LIN {X 0,Y 578.15,Z 1208.915,A -85,B 0,C 180,E1 8907.003,E2 8907.003} C_VEL
LIN {X 0,Y 578.339,Z 1209.667,A -85,B 0,C 180,E1 8911.496,E2 8911.496} C_VEL
LIN {X 0,Y 578.199,Z 1205.911,A -85,B 0,C 180,E1 8916,E2 8916} C_VEL
LIN {X 0,Y 578.472,Z 1197.323,A -85,B 0,C 180,E1 8920.535,E2 8920.535} C_VEL
LIN {X 0,Y 579.28,Z 1182.503,A -85,B 0,C 180,E1 8925.469,E2 8925.469} C_VEL
LIN {X 0,Y 580.832,Z 1163.752,A -85,B 0,C 180,E1 8929.975,E2 8929.975} C_VEL
LIN {X 0,Y 583.523,Z 1139.24,A -85,B 0,C 180,E1 8934.477,E2 8934.477} C_VEL
LIN {X 0,Y 587.576,Z 1110.062,A -85,B 0,C 180,E1 8938.727,E2 8938.727} C_VEL
LIN {X 0,Y 593,Z 1073.863,A -85,B 0,C 180,E1 8942.879,E2 8942.879} C_VEL
LIN {X 0,Y 598.958,Z 1035.476,A -85,B 0,C 180,E1 8946.381,E2 8946.381} C_VEL
LIN {X 0,Y 605.258,Z 993.744,A -85,B 0,C 180,E1 8949.361,E2 8949.361} C_VEL
LIN {X 0,Y 611.066,Z 950.98,A -85,B 0,C 180,E1 8951.738,E2 8951.738} C_VEL
LIN {X 0,Y 616.329,Z 901.945,A -85,B 0,C 180,E1 8953.734,E2 8953.734} C_VEL
LIN {X 0,Y 620.351,Z 854.304,A -85,B 0,C 180,E1 8955.052,E2 8955.052} C_VEL
LIN {X 0,Y 621.032,Z 836.384,A -85,B 0,C 180,E1 8955.439,E2 8955.439} C_VEL
LIN {X 0,Y 598.795,Z 797.154,A -85,B 0,C 180,E1 8958.388,E2 8958.388} C_VEL
LIN {X 0,Y 579.202,Z 767.417,A -85,B 0,C 180,E1 8961.172,E2 8961.172} C_VEL
LIN {X 0,Y 577.121,Z 762.06,A -85,B 0,C 180,E1 8961.632,E2 8961.632} C_VEL
LIN {X 0,Y 577.165,Z 762.06,A -85,B 0,C 180,E1 8966.908,E2 8966.908} C_VEL
LIN {X 0,Y 577.19,Z 762.06,A -85,B 0,C 180,E1 8972.889,E2 8972.889} C_VEL
LIN {X 0,Y 577.361,Z 762.06,A -85,B 0,C 180,E1 8978.499,E2 8978.499} C_VEL
LIN {X 0,Y 577.553,Z 762.06,A -85,B 0,C 180,E1 8983.267,E2 8983.267} C_VEL
LIN {X 0,Y 577.681,Z 762.06,A -85,B 0,C 180,E1 8987.913,E2 8987.913} C_VEL
LIN {X 0,Y 577.909,Z 762.06,A -85,B 0,C 180,E1 8993.988,E2 8993.988} C_VEL
LIN {X 0,Y 578.159,Z 762.06,A -85,B 0,C 180,E1 8999.991,E2 8999.991} C_VEL
LIN {X 0,Y 577.988,Z 762.06,A -85,B 0,C 180,E1 9004.489,E2 9004.489} C_VEL
LIN {X 0,Y 577.816,Z 762.06,A -85,B 0,C 180,E1 9009.018,E2 9009.018} C_VEL
LIN {X 0,Y 577.434,Z 762.06,A -85,B 0,C 180,E1 9014.476,E2 9014.476} C_VEL
LIN {X 0,Y 577.29,Z 762.06,A -85,B 0,C 180,E1 9019.882,E2 9019.882} C_VEL
LIN {X 0,Y 577.282,Z 762.06,A -85,B 0,C 180,E1 9024.747,E2 9024.747} C_VEL
LIN {X 0,Y 577.169,Z 762.06,A -85,B 0,C 180,E1 9030.234,E2 9030.234} C_VEL
LIN {X 0,Y 577.087,Z 762.06,A -85,B 0,C 180,E1 9035.735,E2 9035.735} C_VEL
LIN {X 0,Y 577.062,Z 762.06,A -85,B 0,C 180,E1 9038.874,E2 9038.874} C_VEL
LIN {X 0,Y 579.277,Z 767.544,A -85,B 0,C 180,E1 9039.257,E2 9039.257} C_VEL
LIN {X 0,Y 602.052,Z 802.935,A -85,B 0,C 180,E1 9042.524,E2 9042.524} C_VEL
LIN {X 0,Y 619.608,Z 836.668,A -85,B 0,C 180,E1 9045.179,E2 9045.179} C_VEL
LIN {X 0,Y 615.139,Z 886.033,A -85,B 0,C 180,E1 9046.707,E2 9046.707} C_VEL
LIN {X 0,Y 609.48,Z 932.606,A -85,B 0,C 180,E1 9048.803,E2 9048.803} C_VEL
LIN {X 0,Y 603.473,Z 975.898,A -85,B 0,C 180,E1 9051.376,E2 9051.376} C_VEL
LIN {X 0,Y 597.201,Z 1016.98,A -85,B 0,C 180,E1 9054.547,E2 9054.547} C_VEL
LIN {X 0,Y 591.368,Z 1054.56,A -85,B 0,C 180,E1 9058.196,E2 9058.196} C_VEL
LIN {X 0,Y 586.176,Z 1089.448,A -85,B 0,C 180,E1 9062.497,E2 9062.497} C_VEL
LIN {X 0,Y 582.691,Z 1117.096,A -85,B 0,C 180,E1 9066.804,E2 9066.804} C_VEL
LIN {X 0,Y 580.137,Z 1141.903,A -85,B 0,C 180,E1 9071.787,E2 9071.787} C_VEL
LIN {X 0,Y 578.907,Z 1159.014,A -85,B 0,C 180,E1 9076.414,E2 9076.414} C_VEL
LIN {X 0,Y 578.272,Z 1170.777,A -85,B 0,C 180,E1 9080.98,E2 9080.98} C_VEL
LIN {X 0,Y 578.016,Z 1177.724,A -85,B 0,C 180,E1 9085.502,E2 9085.502} C_VEL
LIN {X 0,Y 578.08,Z 1179.996,A -85,B 0,C 180,E1 9090.001,E2 9090.001} C_VEL
LIN {X 0,Y 578.131,Z 1177.619,A -85,B 0,C 180,E1 9094.498,E2 9094.498} C_VEL
LIN {X 0,Y 578.336,Z 1170.588,A -85,B 0,C 180,E1 9099.02,E2 9099.02} C_VEL
LIN {X 0,Y 578.842,Z 1158.74,A -85,B 0,C 180,E1 9103.59,E2 9103.59} C_VEL
LIN {X 0,Y 580.096,Z 1141.5,A -85,B 0,C 180,E1 9108.216,E2 9108.216} C_VEL
LIN {X 0,Y 582.461,Z 1118.253,A -85,B 0,C 180,E1 9112.903,E2 9112.903} C_VEL
LIN {X 0,Y 586.041,Z 1090.589,A -85,B 0,C 180,E1 9117.256,E2 9117.256} C_VEL
LIN {X 0,Y 591.234,Z 1055.571,A -85,B 0,C 180,E1 9121.599,E2 9121.599} C_VEL
LIN {X 0,Y 596.909,Z 1018.606,A -85,B 0,C 180,E1 9125.225,E2 9125.225} C_VEL
LIN {X 0,Y 603.422,Z 976.128,A -85,B 0,C 180,E1 9128.518,E2 9128.518} C_VEL
LIN {X 0,Y 609.637,Z 932.43,A -85,B 0,C 180,E1 9131.105,E2 9131.105} C_VEL
LIN {X 0,Y 614.684,Z 890.546,A -85,B 0,C 180,E1 9133.017,E2 9133.017} C_VEL
LIN {X 0,Y 619.052,Z 844.789,A -85,B 0,C 180,E1 9134.528,E2 9134.528} C_VEL
LIN {X 0,Y 619.221,Z 836.103,A -85,B 0,C 180,E1 9134.785,E2 9134.785} C_VEL
LIN {X 0,Y 600.743,Z 800.765,A -85,B 0,C 180,E1 9137.568,E2 9137.568} C_VEL
LIN {X 0,Y 579.4,Z 767.603,A -85,B 0,C 180,E1 9140.634,E2 9140.634} C_VEL
LIN {X 0,Y 577.111,Z 762.06,A -85,B 0,C 180,E1 9141.084,E2 9141.084} C_VEL
LIN {X 0,Y 577.121,Z 762.06,A -85,B 0,C 180,E1 9146.918,E2 9146.918} C_VEL
LIN {X 0,Y 577.114,Z 762.06,A -85,B 0,C 180,E1 9152.907,E2 9152.907} C_VEL
LIN {X 0,Y 577.261,Z 762.06,A -85,B 0,C 180,E1 9158.513,E2 9158.513} C_VEL
LIN {X 0,Y 577.429,Z 762.06,A -85,B 0,C 180,E1 9164.84,E2 9164.84} C_VEL
LIN {X 0,Y 577.724,Z 762.06,A -85,B 0,C 180,E1 9169.46,E2 9169.46} C_VEL
LIN {X 0,Y 577.901,Z 762.06,A -85,B 0,C 180,E1 9174.006,E2 9174.006} C_VEL
LIN {X 0,Y 578.06,Z 762.06,A -85,B 0,C 180,E1 9178.511,E2 9178.511} C_VEL
LIN {X 0,Y 577.954,Z 762.06,A -85,B 0,C 180,E1 9183.006,E2 9183.006} C_VEL
LIN {X 0,Y 577.846,Z 762.06,A -85,B 0,C 180,E1 9187.521,E2 9187.521} C_VEL
LIN {X 0,Y 577.677,Z 762.06,A -85,B 0,C 180,E1 9192.087,E2 9192.087} C_VEL
LIN {X 0,Y 577.633,Z 762.06,A -85,B 0,C 180,E1 9196.731,E2 9196.731} C_VEL
LIN {X 0,Y 577.501,Z 762.06,A -85,B 0,C 180,E1 9201.496,E2 9201.496} C_VEL
LIN {X 0,Y 577.334,Z 762.06,A -85,B 0,C 180,E1 9207.136,E2 9207.136} C_VEL
LIN {X 0,Y 577.241,Z 762.06,A -85,B 0,C 180,E1 9213.1,E2 9213.1} C_VEL
LIN {X 0,Y 577.123,Z 762.06,A -85,B 0,C 180,E1 9218.461,E2 9218.461} C_VEL
LIN {X 0,Y 579.443,Z 767.642,A -85,B 0,C 180,E1 9218.865,E2 9218.865} C_VEL
LIN {X 0,Y 602.931,Z 803.858,A -85,B 0,C 180,E1 9222.165,E2 9222.165} C_VEL
LIN {X 0,Y 621.477,Z 837.132,A -85,B 0,C 180,E1 9224.621,E2 9224.621} C_VEL
LIN {X 0,Y 617.556,Z 889.111,A -85,B 0,C 180,E1 9225.855,E2 9225.855} C_VEL
LIN {X 0,Y 613.175,Z 933.192,A -85,B 0,C 180,E1 9227.456,E2 9227.456} C_VEL
LIN {X 0,Y 611.803,Z 944.782,A -85,B 0,C 180,E1 9227.982,E2 9227.982} C_VEL
LIN {X 0,Y 607.308,Z 955.564,A -85,B 0,C 180,E1 9228.234,E2 9228.234} C_VEL
LIN {X 0,Y 602.903,Z 965.984,A -85,B 0,C 180,E1 9228.523,E2 9228.523} C_VEL
LIN {X 0,Y 596.636,Z 1008.633,A -85,B 0,C 180,E1 9231.126,E2 9231.126} C_VEL
LIN {X 0,Y 589.947,Z 1050.374,A -85,B 0,C 180,E1 9234.424,E2 9234.424} C_VEL
LIN {X 0,Y 584.112,Z 1085.938,A -85,B 0,C 180,E1 9237.971,E2 9237.971} C_VEL
LIN {X 0,Y 578.634,Z 1121.078,A -85,B 0,C 180,E1 9242.391,E2 9242.391} C_VEL
LIN {X 0,Y 574.815,Z 1149.399,A -85,B 0,C 180,E1 9246.946,E2 9246.946} C_VEL
LIN {X 0,Y 572.456,Z 1171.697,A -85,B 0,C 180,E1 9251.532,E2 9251.532} C_VEL
LIN {X 0,Y 571.07,Z 1188.871,A -85,B 0,C 180,E1 9256.222,E2 9256.222} C_VEL
LIN {X 0,Y 570.409,Z 1200.678,A -85,B 0,C 180,E1 9260.853,E2 9260.853} C_VEL
LIN {X 0,Y 570.191,Z 1207.667,A -85,B 0,C 180,E1 9265.439,E2 9265.439} C_VEL
LIN {X 0,Y 570.292,Z 1210,A -85,B 0,C 180,E1 9269.999,E2 9269.999} C_VEL
LIN {X 0,Y 570.191,Z 1207.67,A -85,B 0,C 180,E1 9274.559,E2 9274.559} C_VEL
LIN {X 0,Y 570.399,Z 1200.681,A -85,B 0,C 180,E1 9279.145,E2 9279.145} C_VEL
LIN {X 0,Y 571.01,Z 1188.877,A -85,B 0,C 180,E1 9283.778,E2 9283.778} C_VEL
LIN {X 0,Y 572.488,Z 1171.703,A -85,B 0,C 180,E1 9288.465,E2 9288.465} C_VEL
LIN {X 0,Y 575.129,Z 1147.41,A -85,B 0,C 180,E1 9293.415,E2 9293.415} C_VEL
LIN {X 0,Y 578.901,Z 1119.586,A -85,B 0,C 180,E1 9297.812,E2 9297.812} C_VEL
LIN {X 0,Y 584.473,Z 1084.193,A -85,B 0,C 180,E1 9302.224,E2 9302.224} C_VEL
LIN {X 0,Y 590.602,Z 1046.177,A -85,B 0,C 180,E1 9305.943,E2 9305.943} C_VEL
LIN {X 0,Y 597.246,Z 1004.955,A -85,B 0,C 180,E1 9309.134,E2 9309.134} C_VEL
LIN {X 0,Y 603.585,Z 960.631,A -85,B 0,C 180,E1 9311.754,E2 9311.754} C_VEL
LIN {X 0,Y 609.331,Z 913.705,A -85,B 0,C 180,E1 9313.837,E2 9313.837} C_VEL
LIN {X 0,Y 613.929,Z 864.169,A -85,B 0,C 180,E1 9315.339,E2 9315.339} C_VEL
LIN {X 0,Y 615.156,Z 839.358,A -85,B 0,C 180,E1 9315.914,E2 9315.914} C_VEL
LIN {X 0,Y 593.425,Z 801.025,A -85,B 0,C 180,E1 9318.901,E2 9318.901} C_VEL
LIN {X 0,Y 571.54,Z 767.635,A -85,B 0,C 180,E1 9322.125,E2 9322.125} C_VEL
LIN {X 0,Y 569.331,Z 763.533,A -85,B 0,C 180,E1 9322.492,E2 9322.492} C_VEL
LIN {X 0,Y 569.194,Z 762.06,A -85,B 0,C 180,E1 9322.602,E2 9322.602} C_VEL
LIN {X 0,Y 569.21,Z 762.06,A -85,B 0,C 180,E1 9328.158,E2 9328.158} C_VEL
LIN {X 0,Y 569.312,Z 762.06,A -85,B 0,C 180,E1 9333.171,E2 9333.171} C_VEL
LIN {X 0,Y 569.438,Z 762.06,A -85,B 0,C 180,E1 9338.245,E2 9338.245} C_VEL
LIN {X 0,Y 569.61,Z 762.06,A -85,B 0,C 180,E1 9343.026,E2 9343.026} C_VEL
LIN {X 0,Y 569.8,Z 762.06,A -85,B 0,C 180,E1 9348.881,E2 9348.881} C_VEL
LIN {X 0,Y 570.008,Z 762.06,A -85,B 0,C 180,E1 9353.905,E2 9353.905} C_VEL
LIN {X 0,Y 570.259,Z 762.06,A -85,B 0,C 180,E1 9359.991,E2 9359.991} C_VEL
LIN {X 0,Y 570.078,Z 762.06,A -85,B 0,C 180,E1 9364.552,E2 9364.552} C_VEL
LIN {X 0,Y 569.891,Z 762.06,A -85,B 0,C 180,E1 9369.144,E2 9369.144} C_VEL
LIN {X 0,Y 569.572,Z 762.06,A -85,B 0,C 180,E1 9373.803,E2 9373.803} C_VEL
LIN {X 0,Y 569.365,Z 762.06,A -85,B 0,C 180,E1 9380.171,E2 9380.171} C_VEL
LIN {X 0,Y 569.319,Z 762.06,A -85,B 0,C 180,E1 9385.521,E2 9385.521} C_VEL
LIN {X 0,Y 569.271,Z 762.06,A -85,B 0,C 180,E1 9390.274,E2 9390.274} C_VEL
LIN {X 0,Y 569.204,Z 762.06,A -85,B 0,C 180,E1 9395.72,E2 9395.72} C_VEL
LIN {X 0,Y 569.19,Z 762.554,A -85,B 0,C 180,E1 9397.887,E2 9397.887} C_VEL
LIN {X 0,Y 571.828,Z 767.957,A -85,B 0,C 180,E1 9398.335,E2 9398.335} C_VEL
LIN {X 0,Y 595.395,Z 804.724,A -85,B 0,C 180,E1 9401.853,E2 9401.853} C_VEL
LIN {X 0,Y 613.798,Z 839.794,A -85,B 0,C 180,E1 9404.73,E2 9404.73} C_VEL
LIN {X 0,Y 609.147,Z 887.831,A -85,B 0,C 180,E1 9406.252,E2 9406.252} C_VEL
LIN {X 0,Y 603.148,Z 935.142,A -85,B 0,C 180,E1 9408.424,E2 9408.424} C_VEL
LIN {X 0,Y 596.582,Z 979.085,A -85,B 0,C 180,E1 9411.114,E2 9411.114} C_VEL
LIN {X 0,Y 589.91,Z 1020.817,A -85,B 0,C 180,E1 9414.42,E2 9414.42} C_VEL
LIN {X 0,Y 584.051,Z 1056.311,A -85,B 0,C 180,E1 9417.969,E2 9417.969} C_VEL
LIN {X 0,Y 578.578,Z 1091.32,A -85,B 0,C 180,E1 9422.378,E2 9422.378} C_VEL
LIN {X 0,Y 574.813,Z 1119.4,A -85,B 0,C 180,E1 9426.902,E2 9426.902} C_VEL
LIN {X 0,Y 572.368,Z 1141.898,A -85,B 0,C 180,E1 9431.531,E2 9431.531} C_VEL
LIN {X 0,Y 571.071,Z 1159.009,A -85,B 0,C 180,E1 9436.223,E2 9436.223} C_VEL
LIN {X 0,Y 570.386,Z 1170.772,A -85,B 0,C 180,E1 9440.854,E2 9440.854} C_VEL
LIN {X 0,Y 570.117,Z 1177.721,A -85,B 0,C 180,E1 9445.44,E2 9445.44} C_VEL
LIN {X 0,Y 570.179,Z 1179.997,A -85,B 0,C 180,E1 9450.001,E2 9450.001} C_VEL
LIN {X 0,Y 570.228,Z 1177.617,A -85,B 0,C 180,E1 9454.561,E2 9454.561} C_VEL
LIN {X 0,Y 570.439,Z 1170.586,A -85,B 0,C 180,E1 9459.146,E2 9459.146} C_VEL
LIN {X 0,Y 570.998,Z 1158.739,A -85,B 0,C 180,E1 9463.78,E2 9463.78} C_VEL
LIN {X 0,Y 572.335,Z 1141.502,A -85,B 0,C 180,E1 9468.472,E2 9468.472} C_VEL
LIN {X 0,Y 574.916,Z 1118.255,A -85,B 0,C 180,E1 9473.221,E2 9473.221} C_VEL
LIN {X 0,Y 578.709,Z 1090.582,A -85,B 0,C 180,E1 9477.632,E2 9477.632} C_VEL
LIN {X 0,Y 584.177,Z 1055.584,A -85,B 0,C 180,E1 9482.024,E2 9482.024} C_VEL
LIN {X 0,Y 590.194,Z 1018.686,A -85,B 0,C 180,E1 9485.679,E2 9485.679} C_VEL
LIN {X 0,Y 597.13,Z 975.473,A -85,B 0,C 180,E1 9489.056,E2 9489.056} C_VEL
LIN {X 0,Y 604.016,Z 929.667,A -85,B 0,C 180,E1 9491.762,E2 9491.762} C_VEL
LIN {X 0,Y 609.202,Z 888.326,A -85,B 0,C 180,E1 9493.627,E2 9493.627} C_VEL
LIN {X 0,Y 613.553,Z 843.309,A -85,B 0,C 180,E1 9495.091,E2 9495.091} C_VEL
LIN {X 0,Y 612.912,Z 838.347,A -85,B 0,C 180,E1 9495.312,E2 9495.312} C_VEL
LIN {X 0,Y 594.638,Z 803.185,A -85,B 0,C 180,E1 9498.172,E2 9498.172} C_VEL
LIN {X 0,Y 571.59,Z 767.719,A -85,B 0,C 180,E1 9501.605,E2 9501.605} C_VEL
LIN {X 0,Y 569.246,Z 763.044,A -85,B 0,C 180,E1 9502.001,E2 9502.001} C_VEL
LIN {X 0,Y 569.185,Z 762.06,A -85,B 0,C 180,E1 9502.074,E2 9502.074} C_VEL
LIN {X 0,Y 569.212,Z 762.06,A -85,B 0,C 180,E1 9508.161,E2 9508.161} C_VEL
LIN {X 0,Y 569.234,Z 762.06,A -85,B 0,C 180,E1 9513.187,E2 9513.187} C_VEL
LIN {X 0,Y 569.337,Z 762.06,A -85,B 0,C 180,E1 9518.275,E2 9518.275} C_VEL
LIN {X 0,Y 569.488,Z 762.06,A -85,B 0,C 180,E1 9524.624,E2 9524.624} C_VEL
LIN {X 0,Y 569.797,Z 762.06,A -85,B 0,C 180,E1 9529.312,E2 9529.312} C_VEL
LIN {X 0,Y 570.004,Z 762.06,A -85,B 0,C 180,E1 9533.922,E2 9533.922} C_VEL
LIN {X 0,Y 570.161,Z 762.06,A -85,B 0,C 180,E1 9538.49,E2 9538.49} C_VEL
LIN {X 0,Y 570.059,Z 762.06,A -85,B 0,C 180,E1 9543.047,E2 9543.047} C_VEL
LIN {X 0,Y 569.928,Z 762.06,A -85,B 0,C 180,E1 9547.626,E2 9547.626} C_VEL
LIN {X 0,Y 569.78,Z 762.06,A -85,B 0,C 180,E1 9552.257,E2 9552.257} C_VEL
LIN {X 0,Y 569.678,Z 762.06,A -85,B 0,C 180,E1 9557.266,E2 9557.266} C_VEL
LIN {X 0,Y 569.57,Z 762.06,A -85,B 0,C 180,E1 9561.81,E2 9561.81} C_VEL
LIN {X 0,Y 569.451,Z 762.06,A -85,B 0,C 180,E1 9566.822,E2 9566.822} C_VEL
LIN {X 0,Y 569.317,Z 762.06,A -85,B 0,C 180,E1 9572.069,E2 9572.069} C_VEL
LIN {X 0,Y 569.213,Z 762.06,A -85,B 0,C 180,E1 9577.457,E2 9577.457} C_VEL
LIN {X 0,Y 571.505,Z 767.645,A -85,B 0,C 180,E1 9577.876,E2 9577.876} C_VEL
LIN {X 0,Y 593.706,Z 801.317,A -85,B 0,C 180,E1 9581.136,E2 9581.136} C_VEL
LIN {X 0,Y 615.726,Z 840.508,A -85,B 0,C 180,E1 9584.169,E2 9584.169} C_VEL
LIN {X 0,Y 611.568,Z 891.855,A -85,B 0,C 180,E1 9585.422,E2 9585.422} C_VEL
LIN {X 0,Y 606.66,Z 937.336,A -85,B 0,C 180,E1 9587.138,E2 9587.138} C_VEL
LIN {X 0,Y 602.903,Z 965.984,A -85,B 0,C 180,E1 9588.523,E2 9588.523} C_VEL
LIN {X 0,Y 597.769,Z 981.415,A -85,B 0,C 180,E1 9589.145,E2 9589.145} C_VEL
LIN {X 0,Y 592.262,Z 996.481,A -85,B 0,C 180,E1 9589.825,E2 9589.825} C_VEL
LIN {X 0,Y 585.642,Z 1036.578,A -85,B 0,C 180,E1 9592.756,E2 9592.756} C_VEL
LIN {X 0,Y 579.041,Z 1074.678,A -85,B 0,C 180,E1 9596.319,E2 9596.319} C_VEL
LIN {X 0,Y 573.096,Z 1110.074,A -85,B 0,C 180,E1 9600.478,E2 9600.478} C_VEL
LIN {X 0,Y 568.321,Z 1140.428,A -85,B 0,C 180,E1 9605.032,E2 9605.032} C_VEL
LIN {X 0,Y 565.359,Z 1164.734,A -85,B 0,C 180,E1 9609.667,E2 9609.667} C_VEL
LIN {X 0,Y 563.548,Z 1183.702,A -85,B 0,C 180,E1 9614.445,E2 9614.445} C_VEL
LIN {X 0,Y 562.737,Z 1197.314,A -85,B 0,C 180,E1 9619.165,E2 9619.165} C_VEL
LIN {X 0,Y 562.409,Z 1205.908,A -85,B 0,C 180,E1 9623.829,E2 9623.829} C_VEL
LIN {X 0,Y 562.268,Z 1209.666,A -85,B 0,C 180,E1 9628.459,E2 9628.459} C_VEL
LIN {X 0,Y 562.401,Z 1208.911,A -85,B 0,C 180,E1 9633.08,E2 9633.08} C_VEL
LIN {X 0,Y 562.433,Z 1203.551,A -85,B 0,C 180,E1 9637.72,E2 9637.72} C_VEL
LIN {X 0,Y 562.835,Z 1193.421,A -85,B 0,C 180,E1 9642.402,E2 9642.402} C_VEL
LIN {X 0,Y 564.018,Z 1178.003,A -85,B 0,C 180,E1 9647.139,E2 9647.139} C_VEL
LIN {X 0,Y 566.256,Z 1156.978,A -85,B 0,C 180,E1 9651.937,E2 9651.937} C_VEL
LIN {X 0,Y 569.716,Z 1131.625,A -85,B 0,C 180,E1 9656.402,E2 9656.402} C_VEL
LIN {X 0,Y 574.953,Z 1099.018,A -85,B 0,C 180,E1 9660.925,E2 9660.925} C_VEL
LIN {X 0,Y 580.878,Z 1063.701,A -85,B 0,C 180,E1 9664.797,E2 9664.797} C_VEL
LIN {X 0,Y 587.848,Z 1023.085,A -85,B 0,C 180,E1 9668.326,E2 9668.326} C_VEL
LIN {X 0,Y 594.574,Z 981.096,A -85,B 0,C 180,E1 9671.128,E2 9671.128} C_VEL
LIN {X 0,Y 600.97,Z 935.912,A -85,B 0,C 180,E1 9673.434,E2 9673.434} C_VEL
LIN {X 0,Y 605.868,Z 892.707,A -85,B 0,C 180,E1 9675.069,E2 9675.069} C_VEL
LIN {X 0,Y 609.423,Z 842.612,A -85,B 0,C 180,E1 9676.382,E2 9676.382} C_VEL
LIN {X 0,Y 587.325,Z 803.329,A -85,B 0,C 180,E1 9679.54,E2 9679.54} C_VEL
LIN {X 0,Y 563.946,Z 767.982,A -85,B 0,C 180,E1 9683.113,E2 9683.113} C_VEL
LIN {X 0,Y 561.288,Z 762.651,A -85,B 0,C 180,E1 9683.585,E2 9683.585} C_VEL
LIN {X 0,Y 561.297,Z 762.06,A -85,B 0,C 180,E1 9689.484,E2 9689.484} C_VEL
LIN {X 0,Y 561.426,Z 762.06,A -85,B 0,C 180,E1 9694.485,E2 9694.485} C_VEL
LIN {X 0,Y 561.574,Z 762.06,A -85,B 0,C 180,E1 9700.353,E2 9700.353} C_VEL
LIN {X 0,Y 561.786,Z 762.06,A -85,B 0,C 180,E1 9705.983,E2 9705.983} C_VEL
LIN {X 0,Y 561.943,Z 762.06,A -85,B 0,C 180,E1 9710.707,E2 9710.707} C_VEL
LIN {X 0,Y 562.162,Z 762.06,A -85,B 0,C 180,E1 9715.366,E2 9715.366} C_VEL
LIN {X 0,Y 562.358,Z 762.06,A -85,B 0,C 180,E1 9719.991,E2 9719.991} C_VEL
LIN {X 0,Y 562.167,Z 762.06,A -85,B 0,C 180,E1 9724.616,E2 9724.616} C_VEL
LIN {X 0,Y 561.976,Z 762.06,A -85,B 0,C 180,E1 9729.274,E2 9729.274} C_VEL
LIN {X 0,Y 561.615,Z 762.06,A -85,B 0,C 180,E1 9734.391,E2 9734.391} C_VEL
LIN {X 0,Y 561.457,Z 762.06,A -85,B 0,C 180,E1 9740.468,E2 9740.468} C_VEL
LIN {X 0,Y 561.437,Z 762.06,A -85,B 0,C 180,E1 9745.495,E2 9745.495} C_VEL
LIN {X 0,Y 561.345,Z 762.06,A -85,B 0,C 180,E1 9750.747,E2 9750.747} C_VEL
LIN {X 0,Y 561.271,Z 762.06,A -85,B 0,C 180,E1 9756.804,E2 9756.804} C_VEL
LIN {X 0,Y 563.465,Z 767.461,A -85,B 0,C 180,E1 9757.228,E2 9757.228} C_VEL
LIN {X 0,Y 584.428,Z 799.083,A -85,B 0,C 180,E1 9760.503,E2 9760.503} C_VEL
LIN {X 0,Y 605.427,Z 837.685,A -85,B 0,C 180,E1 9763.843,E2 9763.843} C_VEL
LIN {X 0,Y 607.975,Z 843.781,A -85,B 0,C 180,E1 9764.295,E2 9764.295} C_VEL
LIN {X 0,Y 603.011,Z 891.034,A -85,B 0,C 180,E1 9765.845,E2 9765.845} C_VEL
LIN {X 0,Y 596.627,Z 939.154,A -85,B 0,C 180,E1 9768.109,E2 9768.109} C_VEL
LIN {X 0,Y 589.835,Z 981.494,A -85,B 0,C 180,E1 9770.79,E2 9770.79} C_VEL
LIN {X 0,Y 582.949,Z 1022.454,A -85,B 0,C 180,E1 9774.093,E2 9774.093} C_VEL
LIN {X 0,Y 576.73,Z 1058.053,A -85,B 0,C 180,E1 9777.735,E2 9777.735} C_VEL
LIN {X 0,Y 571.242,Z 1091.31,A -85,B 0,C 180,E1 9781.992,E2 9781.992} C_VEL
LIN {X 0,Y 567.324,Z 1118.73,A -85,B 0,C 180,E1 9786.452,E2 9786.452} C_VEL
LIN {X 0,Y 564.619,Z 1141.894,A -85,B 0,C 180,E1 9791.268,E2 9791.268} C_VEL
LIN {X 0,Y 563.23,Z 1159.004,A -85,B 0,C 180,E1 9796.028,E2 9796.028} C_VEL
LIN {X 0,Y 562.499,Z 1170.768,A -85,B 0,C 180,E1 9800.725,E2 9800.725} C_VEL
LIN {X 0,Y 562.437,Z 1175.966,A -85,B 0,C 180,E1 9803.831,E2 9803.831} C_VEL
LIN {X 0,Y 562.183,Z 1179.677,A -85,B 0,C 180,E1 9808.461,E2 9808.461} C_VEL
LIN {X 0,Y 562.281,Z 1178.879,A -85,B 0,C 180,E1 9813.082,E2 9813.082} C_VEL
LIN {X 0,Y 562.525,Z 1173.478,A -85,B 0,C 180,E1 9817.72,E2 9817.72} C_VEL
LIN {X 0,Y 562.924,Z 1163.291,A -85,B 0,C 180,E1 9822.402,E2 9822.402} C_VEL
LIN {X 0,Y 564.173,Z 1146.746,A -85,B 0,C 180,E1 9827.42,E2 9827.42} C_VEL
LIN {X 0,Y 566.414,Z 1125.084,A -85,B 0,C 180,E1 9832.281,E2 9832.281} C_VEL
LIN {X 0,Y 570.284,Z 1097.463,A -85,B 0,C 180,E1 9836.997,E2 9836.997} C_VEL
LIN {X 0,Y 575.235,Z 1066.923,A -85,B 0,C 180,E1 9841.147,E2 9841.147} C_VEL
LIN {X 0,Y 581.851,Z 1028.484,A -85,B 0,C 180,E1 9845.251,E2 9845.251} C_VEL
LIN {X 0,Y 588.487,Z 990.042,A -85,B 0,C 180,E1 9848.498,E2 9848.498} C_VEL
LIN {X 0,Y 595.3,Z 947.817,A -85,B 0,C 180,E1 9851.3,E2 9851.3} C_VEL
LIN {X 0,Y 601.595,Z 903.185,A -85,B 0,C 180,E1 9853.566,E2 9853.566} C_VEL
LIN {X 0,Y 607.022,Z 853.16,A -85,B 0,C 180,E1 9855.359,E2 9855.359} C_VEL
LIN {X 0,Y 607.554,Z 842.684,A -85,B 0,C 180,E1 9855.692,E2 9855.692} C_VEL
LIN {X 0,Y 590.505,Z 809.049,A -85,B 0,C 180,E1 9858.493,E2 9858.493} C_VEL
LIN {X 0,Y 567.8,Z 773.747,A -85,B 0,C 180,E1 9861.973,E2 9861.973} C_VEL
LIN {X 0,Y 563.437,Z 767.429,A -85,B 0,C 180,E1 9862.68,E2 9862.68} C_VEL
LIN {X 0,Y 561.288,Z 762.06,A -85,B 0,C 180,E1 9863.153,E2 9863.153} C_VEL
LIN {X 0,Y 561.273,Z 762.06,A -85,B 0,C 180,E1 9869.491,E2 9869.491} C_VEL
LIN {X 0,Y 561.345,Z 762.06,A -85,B 0,C 180,E1 9874.501,E2 9874.501} C_VEL
LIN {X 0,Y 561.377,Z 762.06,A -85,B 0,C 180,E1 9880.414,E2 9880.414} C_VEL
LIN {X 0,Y 561.651,Z 762.06,A -85,B 0,C 180,E1 9885.998,E2 9885.998} C_VEL
LIN {X 0,Y 561.992,Z 762.06,A -85,B 0,C 180,E1 9890.726,E2 9890.726} C_VEL
LIN {X 0,Y 562.285,Z 762.06,A -85,B 0,C 180,E1 9896.928,E2 9896.928} C_VEL
LIN {X 0,Y 562.311,Z 762.06,A -85,B 0,C 180,E1 9901.549,E2 9901.549} C_VEL
LIN {X 0,Y 562.115,Z 762.06,A -85,B 0,C 180,E1 9906.181,E2 9906.181} C_VEL
LIN {X 0,Y 561.914,Z 762.06,A -85,B 0,C 180,E1 9910.858,E2 9910.858} C_VEL
LIN {X 0,Y 561.791,Z 762.06,A -85,B 0,C 180,E1 9915.611,E2 9915.611} C_VEL
LIN {X 0,Y 561.702,Z 762.06,A -85,B 0,C 180,E1 9920.478,E2 9920.478} C_VEL
LIN {X 0,Y 561.558,Z 762.06,A -85,B 0,C 180,E1 9925.509,E2 9925.509} C_VEL
LIN {X 0,Y 561.426,Z 762.06,A -85,B 0,C 180,E1 9930.763,E2 9930.763} C_VEL
LIN {X 0,Y 561.308,Z 762.128,A -85,B 0,C 180,E1 9936.413,E2 9936.413} C_VEL
LIN {X 0,Y 563.528,Z 767.57,A -85,B 0,C 180,E1 9936.828,E2 9936.828} C_VEL
LIN {X 0,Y 581.473,Z 794.059,A -85,B 0,C 180,E1 9939.612,E2 9939.612} C_VEL
LIN {X 0,Y 604.48,Z 832.907,A -85,B 0,C 180,E1 9942.882,E2 9942.882} C_VEL
LIN {X 0,Y 609.987,Z 843.742,A -85,B 0,C 180,E1 9943.703,E2 9943.703} C_VEL
LIN {X 0,Y 605.712,Z 893.539,A -85,B 0,C 180,E1 9944.948,E2 9944.948} C_VEL
LIN {X 0,Y 600.463,Z 939.105,A -85,B 0,C 180,E1 9946.704,E2 9946.704} C_VEL
LIN {X 0,Y 594.099,Z 984.295,A -85,B 0,C 180,E1 9949.057,E2 9949.057} C_VEL
LIN {X 0,Y 592.262,Z 996.481,A -85,B 0,C 180,E1 9949.825,E2 9949.825} C_VEL
LIN {X 0,Y 586.613,Z 1011.277,A -85,B 0,C 180,E1 9950.564,E2 9950.564} C_VEL
LIN {X 0,Y 580.867,Z 1025.602,A -85,B 0,C 180,E1 9951.376,E2 9951.376} C_VEL
LIN {X 0,Y 573.609,Z 1067.035,A -85,B 0,C 180,E1 9955.063,E2 9955.063} C_VEL
LIN {X 0,Y 567.199,Z 1102.455,A -85,B 0,C 180,E1 9959.084,E2 9959.084} C_VEL
LIN {X 0,Y 561.943,Z 1134.398,A -85,B 0,C 180,E1 9963.659,E2 9963.659} C_VEL
LIN {X 0,Y 558.118,Z 1161.32,A -85,B 0,C 180,E1 9968.656,E2 9968.656} C_VEL
LIN {X 0,Y 555.975,Z 1181.012,A -85,B 0,C 180,E1 9973.417,E2 9973.417} C_VEL
LIN {X 0,Y 554.918,Z 1195.114,A -85,B 0,C 180,E1 9978.101,E2 9978.101} C_VEL
LIN {X 0,Y 554.551,Z 1204.752,A -85,B 0,C 180,E1 9982.956,E2 9982.956} C_VEL
LIN {X 0,Y 554.473,Z 1208.906,A -85,B 0,C 180,E1 9986.875,E2 9986.875} C_VEL
LIN {X 0,Y 554.65,Z 1209.667,A -85,B 0,C 180,E1 9991.56,E2 9991.56} C_VEL
LIN {X 0,Y 554.552,Z 1205.911,A -85,B 0,C 180,E1 9996.257,E2 9996.257} C_VEL
LIN {X 0,Y 554.854,Z 1197.314,A -85,B 0,C 180,E1 10000.989,E2 10000.989} C_VEL
LIN {X 0,Y 555.743,Z 1183.708,A -85,B 0,C 180,E1 10005.777,E2 10005.777} C_VEL
LIN {X 0,Y 557.689,Z 1164.737,A -85,B 0,C 180,E1 10010.624,E2 10010.624} C_VEL
LIN {X 0,Y 560.856,Z 1140.432,A -85,B 0,C 180,E1 10015.322,E2 10015.322} C_VEL
LIN {X 0,Y 565.956,Z 1110.044,A -85,B 0,C 180,E1 10019.936,E2 10019.936} C_VEL
LIN {X 0,Y 572.132,Z 1074.775,A -85,B 0,C 180,E1 10024.132,E2 10024.132} C_VEL
LIN {X 0,Y 578.924,Z 1037.519,A -85,B 0,C 180,E1 10027.663,E2 10027.663} C_VEL
LIN {X 0,Y 586.201,Z 995.009,A -85,B 0,C 180,E1 10030.772,E2 10030.772} C_VEL
LIN {X 0,Y 592.787,Z 952.278,A -85,B 0,C 180,E1 10033.203,E2 10033.203} C_VEL
LIN {X 0,Y 598.625,Z 905.735,A -85,B 0,C 180,E1 10035.168,E2 10035.168} C_VEL
LIN {X 0,Y 603.579,Z 855.118,A -85,B 0,C 180,E1 10036.623,E2 10036.623} C_VEL
LIN {X 0,Y 603.757,Z 845.97,A -85,B 0,C 180,E1 10036.852,E2 10036.852} C_VEL
LIN {X 0,Y 582.596,Z 808.035,A -85,B 0,C 180,E1 10039.997,E2 10039.997} C_VEL
LIN {X 0,Y 560.294,Z 774.157,A -85,B 0,C 180,E1 10043.48,E2 10043.48} C_VEL
LIN {X 0,Y 555.639,Z 767.63,A -85,B 0,C 180,E1 10044.268,E2 10044.268} C_VEL
LIN {X 0,Y 553.345,Z 762.06,A -85,B 0,C 180,E1 10044.793,E2 10044.793} C_VEL
LIN {X 0,Y 553.428,Z 762.06,A -85,B 0,C 180,E1 10050.895,E2 10050.895} C_VEL
LIN {X 0,Y 553.481,Z 762.06,A -85,B 0,C 180,E1 10055.818,E2 10055.818} C_VEL
LIN {X 0,Y 553.688,Z 762.06,A -85,B 0,C 180,E1 10060.876,E2 10060.876} C_VEL
LIN {X 0,Y 553.88,Z 762.06,A -85,B 0,C 180,E1 10065.779,E2 10065.779} C_VEL
LIN {X 0,Y 554.024,Z 762.06,A -85,B 0,C 180,E1 10070.573,E2 10070.573} C_VEL
LIN {X 0,Y 554.283,Z 762.06,A -85,B 0,C 180,E1 10075.3,E2 10075.3} C_VEL
LIN {X 0,Y 554.481,Z 762.06,A -85,B 0,C 180,E1 10079.991,E2 10079.991} C_VEL
LIN {X 0,Y 554.289,Z 762.06,A -85,B 0,C 180,E1 10084.682,E2 10084.682} C_VEL
LIN {X 0,Y 554.05,Z 762.06,A -85,B 0,C 180,E1 10089.408,E2 10089.408} C_VEL
LIN {X 0,Y 553.741,Z 762.06,A -85,B 0,C 180,E1 10094.206,E2 10094.206} C_VEL
LIN {X 0,Y 553.507,Z 762.06,A -85,B 0,C 180,E1 10099.112,E2 10099.112} C_VEL
LIN {X 0,Y 553.482,Z 762.06,A -85,B 0,C 180,E1 10104.162,E2 10104.162} C_VEL
LIN {X 0,Y 553.458,Z 762.06,A -85,B 0,C 180,E1 10109.422,E2 10109.422} C_VEL
LIN {X 0,Y 553.334,Z 762.06,A -85,B 0,C 180,E1 10115.685,E2 10115.685} C_VEL
LIN {X 0,Y 555.596,Z 767.546,A -85,B 0,C 180,E1 10116.14,E2 10116.14} C_VEL
LIN {X 0,Y 558.258,Z 771.147,A -85,B 0,C 180,E1 10116.592,E2 10116.592} C_VEL
LIN {X 0,Y 580.66,Z 805.425,A -85,B 0,C 180,E1 10120.204,E2 10120.204} C_VEL
LIN {X 0,Y 600.767,Z 843.329,A -85,B 0,C 180,E1 10123.561,E2 10123.561} C_VEL
LIN {X 0,Y 602.173,Z 847.888,A -85,B 0,C 180,E1 10123.862,E2 10123.862} C_VEL
LIN {X 0,Y 596.52,Z 897.405,A -85,B 0,C 180,E1 10125.56,E2 10125.56} C_VEL
LIN {X 0,Y 590.116,Z 942.621,A -85,B 0,C 180,E1 10127.766,E2 10127.766} C_VEL
LIN {X 0,Y 582.583,Z 987.13,A -85,B 0,C 180,E1 10130.678,E2 10130.678} C_VEL
LIN {X 0,Y 575.463,Z 1026.767,A -85,B 0,C 180,E1 10134.018,E2 10134.018} C_VEL
LIN {X 0,Y 568.529,Z 1064.895,A -85,B 0,C 180,E1 10138.094,E2 10138.094} C_VEL
LIN {X 0,Y 563.215,Z 1095.76,A -85,B 0,C 180,E1 10142.267,E2 10142.267} C_VEL
LIN {X 0,Y 559.004,Z 1124.503,A -85,B 0,C 180,E1 10147.205,E2 10147.205} C_VEL
LIN {X 0,Y 556.466,Z 1146.6,A -85,B 0,C 180,E1 10152.202,E2 10152.202} C_VEL
LIN {X 0,Y 555.106,Z 1162.435,A -85,B 0,C 180,E1 10157.023,E2 10157.023} C_VEL
LIN {X 0,Y 554.59,Z 1172.307,A -85,B 0,C 180,E1 10161.382,E2 10161.382} C_VEL
LIN {X 0,Y 554.342,Z 1177.714,A -85,B 0,C 180,E1 10165.31,E2 10165.31} C_VEL
LIN {X 0,Y 554.398,Z 1179.997,A -85,B 0,C 180,E1 10170.001,E2 10170.001} C_VEL
LIN {X 0,Y 554.442,Z 1177.612,A -85,B 0,C 180,E1 10174.691,E2 10174.691} C_VEL
LIN {X 0,Y 554.653,Z 1170.583,A -85,B 0,C 180,E1 10179.409,E2 10179.409} C_VEL
LIN {X 0,Y 555.342,Z 1158.736,A -85,B 0,C 180,E1 10184.176,E2 10184.176} C_VEL
LIN {X 0,Y 556.878,Z 1141.505,A -85,B 0,C 180,E1 10189.004,E2 10189.004} C_VEL
LIN {X 0,Y 559.83,Z 1118.259,A -85,B 0,C 180,E1 10193.885,E2 10193.885} C_VEL
LIN {X 0,Y 564.093,Z 1090.93,A -85,B 0,C 180,E1 10198.361,E2 10198.361} C_VEL
LIN {X 0,Y 570.141,Z 1056.032,A -85,B 0,C 180,E1 10202.854,E2 10202.854} C_VEL
LIN {X 0,Y 576.811,Z 1019.243,A -85,B 0,C 180,E1 10206.584,E2 10206.584} C_VEL
LIN {X 0,Y 584.514,Z 976.286,A -85,B 0,C 180,E1 10210.026,E2 10210.026} C_VEL
LIN {X 0,Y 591.602,Z 933.761,A -85,B 0,C 180,E1 10212.611,E2 10212.611} C_VEL
LIN {X 0,Y 597.431,Z 891.395,A -85,B 0,C 180,E1 10214.58,E2 10214.58} C_VEL
LIN {X 0,Y 601.795,Z 845.89,A -85,B 0,C 180,E1 10216.16,E2 10216.16} C_VEL
LIN {X 0,Y 585.029,Z 812.878,A -85,B 0,C 180,E1 10219,E2 10219} C_VEL
LIN {X 0,Y 564.055,Z 779.703,A -85,B 0,C 180,E1 10222.344,E2 10222.344} C_VEL
LIN {X 0,Y 555.819,Z 767.759,A -85,B 0,C 180,E1 10223.725,E2 10223.725} C_VEL
LIN {X 0,Y 553.44,Z 763.354,A -85,B 0,C 180,E1 10224.162,E2 10224.162} C_VEL
LIN {X 0,Y 553.313,Z 762.06,A -85,B 0,C 180,E1 10224.261,E2 10224.261} C_VEL
LIN {X 0,Y 553.288,Z 762.06,A -85,B 0,C 180,E1 10228.755,E2 10228.755} C_VEL
LIN {X 0,Y 553.411,Z 762.06,A -85,B 0,C 180,E1 10234.302,E2 10234.302} C_VEL
LIN {X 0,Y 553.453,Z 762.06,A -85,B 0,C 180,E1 10239.222,E2 10239.222} C_VEL
LIN {X 0,Y 553.619,Z 762.06,A -85,B 0,C 180,E1 10244.172,E2 10244.172} C_VEL
LIN {X 0,Y 553.971,Z 762.06,A -85,B 0,C 180,E1 10249.117,E2 10249.117} C_VEL
LIN {X 0,Y 554.192,Z 762.06,A -85,B 0,C 180,E1 10253.748,E2 10253.748} C_VEL
LIN {X 0,Y 554.366,Z 762.06,A -85,B 0,C 180,E1 10258.447,E2 10258.447} C_VEL
LIN {X 0,Y 554.25,Z 762.06,A -85,B 0,C 180,E1 10263.134,E2 10263.134} C_VEL
LIN {X 0,Y 554.108,Z 762.06,A -85,B 0,C 180,E1 10267.845,E2 10267.845} C_VEL
LIN {X 0,Y 553.946,Z 762.06,A -85,B 0,C 180,E1 10272.613,E2 10272.613} C_VEL
LIN {X 0,Y 553.848,Z 762.06,A -85,B 0,C 180,E1 10277.472,E2 10277.472} C_VEL
LIN {X 0,Y 553.695,Z 762.06,A -85,B 0,C 180,E1 10282.469,E2 10282.469} C_VEL
LIN {X 0,Y 553.572,Z 762.06,A -85,B 0,C 180,E1 10287.656,E2 10287.656} C_VEL
LIN {X 0,Y 553.417,Z 762.06,A -85,B 0,C 180,E1 10293.106,E2 10293.106} C_VEL
LIN {X 0,Y 553.396,Z 762.585,A -85,B 0,C 180,E1 10295.308,E2 10295.308} C_VEL
LIN {X 0,Y 555.901,Z 767.849,A -85,B 0,C 180,E1 10295.781,E2 10295.781} C_VEL
LIN {X 0,Y 570.852,Z 789.719,A -85,B 0,C 180,E1 10298.231,E2 10298.231} C_VEL
LIN {X 0,Y 593.123,Z 825.84,A -85,B 0,C 180,E1 10301.55,E2 10301.55} C_VEL
LIN {X 0,Y 604.231,Z 848.157,A -85,B 0,C 180,E1 10303.253,E2 10303.253} C_VEL
LIN {X 0,Y 599.739,Z 896.16,A -85,B 0,C 180,E1 10304.502,E2 10304.502} C_VEL
LIN {X 0,Y 594.07,Z 942.705,A -85,B 0,C 180,E1 10306.347,E2 10306.347} C_VEL
LIN {X 0,Y 587.369,Z 987.767,A -85,B 0,C 180,E1 10308.756,E2 10308.756} C_VEL
LIN {X 0,Y 580.867,Z 1025.602,A -85,B 0,C 180,E1 10311.376,E2 10311.376} C_VEL
LIN {X 0,Y 575.227,Z 1039.724,A -85,B 0,C 180,E1 10312.281,E2 10312.281} C_VEL
LIN {X 0,Y 569.498,Z 1053.121,A -85,B 0,C 180,E1 10313.225,E2 10313.225} C_VEL
LIN {X 0,Y 562.387,Z 1090.198,A -85,B 0,C 180,E1 10317.136,E2 10317.136} C_VEL
LIN {X 0,Y 556.562,Z 1121.992,A -85,B 0,C 180,E1 10321.336,E2 10321.336} C_VEL
LIN {X 0,Y 551.958,Z 1150.381,A -85,B 0,C 180,E1 10326.128,E2 10326.128} C_VEL
LIN {X 0,Y 549.042,Z 1173.465,A -85,B 0,C 180,E1 10331.153,E2 10331.153} C_VEL
LIN {X 0,Y 547.372,Z 1191.152,A -85,B 0,C 180,E1 10336.428,E2 10336.428} C_VEL
LIN {X 0,Y 546.735,Z 1202.219,A -85,B 0,C 180,E1 10341.256,E2 10341.256} C_VEL
LIN {X 0,Y 546.511,Z 1207.659,A -85,B 0,C 180,E1 10345.241,E2 10345.241} C_VEL
LIN {X 0,Y 546.612,Z 1210,A -85,B 0,C 180,E1 10349.999,E2 10349.999} C_VEL
LIN {X 0,Y 546.513,Z 1207.661,A -85,B 0,C 180,E1 10354.757,E2 10354.757} C_VEL
LIN {X 0,Y 546.777,Z 1200.672,A -85,B 0,C 180,E1 10359.544,E2 10359.544} C_VEL
LIN {X 0,Y 547.655,Z 1187.874,A -85,B 0,C 180,E1 10364.723,E2 10364.723} C_VEL
LIN {X 0,Y 549.362,Z 1169.981,A -85,B 0,C 180,E1 10369.687,E2 10369.687} C_VEL
LIN {X 0,Y 552.556,Z 1146.562,A -85,B 0,C 180,E1 10374.599,E2 10374.599} C_VEL
LIN {X 0,Y 557.232,Z 1118.122,A -85,B 0,C 180,E1 10379.217,E2 10379.217} C_VEL
LIN {X 0,Y 563.679,Z 1083.444,A -85,B 0,C 180,E1 10383.664,E2 10383.664} C_VEL
LIN {X 0,Y 570.73,Z 1046.04,A -85,B 0,C 180,E1 10387.405,E2 10387.405} C_VEL
LIN {X 0,Y 578.352,Z 1004.421,A -85,B 0,C 180,E1 10390.669,E2 10390.669} C_VEL
LIN {X 0,Y 585.91,Z 958.038,A -85,B 0,C 180,E1 10393.435,E2 10393.435} C_VEL
LIN {X 0,Y 592.346,Z 910.765,A -85,B 0,C 180,E1 10395.536,E2 10395.536} C_VEL
LIN {X 0,Y 597.761,Z 858.834,A -85,B 0,C 180,E1 10397.083,E2 10397.083} C_VEL
LIN {X 0,Y 598.044,Z 849.194,A -85,B 0,C 180,E1 10397.345,E2 10397.345} C_VEL
LIN {X 0,Y 576.5,Z 810.22,A -85,B 0,C 180,E1 10400.676,E2 10400.676} C_VEL
LIN {X 0,Y 552.981,Z 774.745,A -85,B 0,C 180,E1 10404.495,E2 10404.495} C_VEL
LIN {X 0,Y 547.788,Z 767.725,A -85,B 0,C 180,E1 10405.415,E2 10405.415} C_VEL
LIN {X 0,Y 545.421,Z 762.988,A -85,B 0,C 180,E1 10405.883,E2 10405.883} C_VEL
LIN {X 0,Y 545.369,Z 762.06,A -85,B 0,C 180,E1 10406.225,E2 10406.225} C_VEL
LIN {X 0,Y 545.545,Z 762.06,A -85,B 0,C 180,E1 10412.419,E2 10412.419} C_VEL
LIN {X 0,Y 545.588,Z 762.06,A -85,B 0,C 180,E1 10417.178,E2 10417.178} C_VEL
LIN {X 0,Y 545.824,Z 762.06,A -85,B 0,C 180,E1 10422.263,E2 10422.263} C_VEL
LIN {X 0,Y 546.011,Z 762.06,A -85,B 0,C 180,E1 10427.201,E2 10427.201} C_VEL
LIN {X 0,Y 546.191,Z 762.06,A -85,B 0,C 180,E1 10432.04,E2 10432.04} C_VEL
LIN {X 0,Y 546.334,Z 762.06,A -85,B 0,C 180,E1 10436.82,E2 10436.82} C_VEL
LIN {X 0,Y 546.452,Z 762.06,A -85,B 0,C 180,E1 10441.575,E2 10441.575} C_VEL
LIN {X 0,Y 546.315,Z 762.06,A -85,B 0,C 180,E1 10446.342,E2 10446.342} C_VEL
LIN {X 0,Y 546.02,Z 762.06,A -85,B 0,C 180,E1 10451.159,E2 10451.159} C_VEL
LIN {X 0,Y 545.682,Z 762.06,A -85,B 0,C 180,E1 10456.065,E2 10456.065} C_VEL
LIN {X 0,Y 545.624,Z 762.06,A -85,B 0,C 180,E1 10461.09,E2 10461.09} C_VEL
LIN {X 0,Y 545.547,Z 762.06,A -85,B 0,C 180,E1 10466.293,E2 10466.293} C_VEL
LIN {X 0,Y 545.44,Z 762.06,A -85,B 0,C 180,E1 10471.746,E2 10471.746} C_VEL
LIN {X 0,Y 545.404,Z 762.442,A -85,B 0,C 180,E1 10474.519,E2 10474.519} C_VEL
LIN {X 0,Y 547.937,Z 767.829,A -85,B 0,C 180,E1 10475.027,E2 10475.027} C_VEL
LIN {X 0,Y 563.215,Z 790.003,A -85,B 0,C 180,E1 10477.661,E2 10477.661} C_VEL
LIN {X 0,Y 583.043,Z 823.012,A -85,B 0,C 180,E1 10480.975,E2 10480.975} C_VEL
LIN {X 0,Y 596.462,Z 850.651,A -85,B 0,C 180,E1 10483.39,E2 10483.39} C_VEL
LIN {X 0,Y 590.61,Z 899.461,A -85,B 0,C 180,E1 10485.093,E2 10485.093} C_VEL
LIN {X 0,Y 583.984,Z 943.939,A -85,B 0,C 180,E1 10487.297,E2 10487.297} C_VEL
LIN {X 0,Y 576.09,Z 988.614,A -85,B 0,C 180,E1 10490.256,E2 10490.256} C_VEL
LIN {X 0,Y 568.766,Z 1026.97,A -85,B 0,C 180,E1 10493.55,E2 10493.55} C_VEL
LIN {X 0,Y 561.543,Z 1064.887,A -85,B 0,C 180,E1 10497.649,E2 10497.649} C_VEL
LIN {X 0,Y 555.891,Z 1095.753,A -85,B 0,C 180,E1 10501.869,E2 10501.869} C_VEL
LIN {X 0,Y 551.371,Z 1124.827,A -85,B 0,C 180,E1 10506.936,E2 10506.936} C_VEL
LIN {X 0,Y 548.695,Z 1146.596,A -85,B 0,C 180,E1 10511.941,E2 10511.941} C_VEL
LIN {X 0,Y 547.267,Z 1162.43,A -85,B 0,C 180,E1 10516.833,E2 10516.833} C_VEL
LIN {X 0,Y 546.721,Z 1172.306,A -85,B 0,C 180,E1 10521.257,E2 10521.257} C_VEL
LIN {X 0,Y 546.444,Z 1177.71,A -85,B 0,C 180,E1 10525.242,E2 10525.242} C_VEL
LIN {X 0,Y 546.497,Z 1179.997,A -85,B 0,C 180,E1 10530.001,E2 10530.001} C_VEL
LIN {X 0,Y 546.54,Z 1177.61,A -85,B 0,C 180,E1 10534.759,E2 10534.759} C_VEL
LIN {X 0,Y 546.781,Z 1170.582,A -85,B 0,C 180,E1 10539.546,E2 10539.546} C_VEL
LIN {X 0,Y 547.514,Z 1158.735,A -85,B 0,C 180,E1 10544.383,E2 10544.383} C_VEL
LIN {X 0,Y 549.158,Z 1141.506,A -85,B 0,C 180,E1 10549.282,E2 10549.282} C_VEL
LIN {X 0,Y 552.514,Z 1117.244,A -85,B 0,C 180,E1 10554.423,E2 10554.423} C_VEL
LIN {X 0,Y 557.013,Z 1089.663,A -85,B 0,C 180,E1 10558.949,E2 10558.949} C_VEL
LIN {X 0,Y 563.332,Z 1055.369,A -85,B 0,C 180,E1 10563.39,E2 10563.39} C_VEL
LIN {X 0,Y 570.635,Z 1016.979,A -85,B 0,C 180,E1 10567.293,E2 10567.293} C_VEL
LIN {X 0,Y 578.527,Z 975.459,A -85,B 0,C 180,E1 10570.622,E2 10570.622} C_VEL
LIN {X 0,Y 586.196,Z 930.418,A -85,B 0,C 180,E1 10573.343,E2 10573.343} C_VEL
LIN {X 0,Y 592.361,Z 887.657,A -85,B 0,C 180,E1 10575.281,E2 10575.281} C_VEL
LIN {X 0,Y 596.007,Z 849.089,A -85,B 0,C 180,E1 10576.631,E2 10576.631} C_VEL
LIN {X 0,Y 578.652,Z 814.759,A -85,B 0,C 180,E1 10579.687,E2 10579.687} C_VEL
LIN {X 0,Y 556.886,Z 780.5,A -85,B 0,C 180,E1 10583.303,E2 10583.303} C_VEL
LIN {X 0,Y 547.997,Z 767.88,A -85,B 0,C 180,E1 10584.863,E2 10584.863} C_VEL
LIN {X 0,Y 545.419,Z 762.703,A -85,B 0,C 180,E1 10585.372,E2 10585.372} C_VEL
LIN {X 0,Y 545.374,Z 762.06,A -85,B 0,C 180,E1 10590.098,E2 10590.098} C_VEL
LIN {X 0,Y 545.507,Z 762.06,A -85,B 0,C 180,E1 10596.085,E2 10596.085} C_VEL
LIN {X 0,Y 545.602,Z 762.06,A -85,B 0,C 180,E1 10602.274,E2 10602.274} C_VEL
LIN {X 0,Y 545.939,Z 762.06,A -85,B 0,C 180,E1 10607.218,E2 10607.218} C_VEL
LIN {X 0,Y 546.223,Z 762.06,A -85,B 0,C 180,E1 10613.12,E2 10613.12} C_VEL
LIN {X 0,Y 546.464,Z 762.06,A -85,B 0,C 180,E1 10618.425,E2 10618.425} C_VEL
LIN {X 0,Y 546.345,Z 762.06,A -85,B 0,C 180,E1 10623.18,E2 10623.18} C_VEL
LIN {X 0,Y 546.205,Z 762.06,A -85,B 0,C 180,E1 10627.959,E2 10627.959} C_VEL
LIN {X 0,Y 546.019,Z 762.06,A -85,B 0,C 180,E1 10632.799,E2 10632.799} C_VEL
LIN {X 0,Y 545.918,Z 762.06,A -85,B 0,C 180,E1 10637.734,E2 10637.734} C_VEL
LIN {X 0,Y 545.742,Z 762.06,A -85,B 0,C 180,E1 10642.815,E2 10642.815} C_VEL
LIN {X 0,Y 545.654,Z 762.06,A -85,B 0,C 180,E1 10648.092,E2 10648.092} C_VEL
LIN {X 0,Y 545.458,Z 762.698,A -85,B 0,C 180,E1 10654.127,E2 10654.127} C_VEL
LIN {X 0,Y 548.031,Z 767.874,A -85,B 0,C 180,E1 10654.635,E2 10654.635} C_VEL
LIN {X 0,Y 566.313,Z 794.344,A -85,B 0,C 180,E1 10657.743,E2 10657.743} C_VEL
LIN {X 0,Y 589.21,Z 832.077,A -85,B 0,C 180,E1 10661.257,E2 10661.257} C_VEL
LIN {X 0,Y 598.614,Z 850.551,A -85,B 0,C 180,E1 10662.75,E2 10662.75} C_VEL
LIN {X 0,Y 593.803,Z 898.592,A -85,B 0,C 180,E1 10664.042,E2 10664.042} C_VEL
LIN {X 0,Y 587.841,Z 945.406,A -85,B 0,C 180,E1 10665.942,E2 10665.942} C_VEL
LIN {X 0,Y 580.914,Z 989.284,A -85,B 0,C 180,E1 10668.34,E2 10668.34} C_VEL
LIN {X 0,Y 573.008,Z 1033.563,A -85,B 0,C 180,E1 10671.527,E2 10671.527} C_VEL
LIN {X 0,Y 569.498,Z 1053.121,A -85,B 0,C 180,E1 10673.225,E2 10673.225} C_VEL
LIN {X 0,Y 563.591,Z 1066.22,A -85,B 0,C 180,E1 10674.247,E2 10674.247} C_VEL
LIN {X 0,Y 557.762,Z 1078.73,A -85,B 0,C 180,E1 10675.351,E2 10675.351} C_VEL
LIN {X 0,Y 551.364,Z 1111.274,A -85,B 0,C 180,E1 10679.375,E2 10679.375} C_VEL
LIN {X 0,Y 545.953,Z 1141.011,A -85,B 0,C 180,E1 10684.042,E2 10684.042} C_VEL
LIN {X 0,Y 542.374,Z 1164.738,A -85,B 0,C 180,E1 10688.764,E2 10688.764} C_VEL
LIN {X 0,Y 540.121,Z 1183.699,A -85,B 0,C 180,E1 10693.753,E2 10693.753} C_VEL
LIN {X 0,Y 539.093,Z 1197.686,A -85,B 0,C 180,E1 10698.846,E2 10698.846} C_VEL
LIN {X 0,Y 538.762,Z 1205.908,A -85,B 0,C 180,E1 10703.558,E2 10703.558} C_VEL
LIN {X 0,Y 538.575,Z 1209.666,A -85,B 0,C 180,E1 10708.391,E2 10708.391} C_VEL
LIN {X 0,Y 538.867,Z 1209.667,A -85,B 0,C 180,E1 10711.606,E2 10711.606} C_VEL
LIN {X 0,Y 538.765,Z 1205.911,A -85,B 0,C 180,E1 10716.441,E2 10716.441} C_VEL
LIN {X 0,Y 539.106,Z 1197.308,A -85,B 0,C 180,E1 10721.315,E2 10721.315} C_VEL
LIN {X 0,Y 540.118,Z 1183.706,A -85,B 0,C 180,E1 10726.246,E2 10726.246} C_VEL
LIN {X 0,Y 542.358,Z 1164.74,A -85,B 0,C 180,E1 10731.235,E2 10731.235} C_VEL
LIN {X 0,Y 546.283,Z 1139.229,A -85,B 0,C 180,E1 10736.268,E2 10736.268} C_VEL
LIN {X 0,Y 551.696,Z 1109.569,A -85,B 0,C 180,E1 10740.86,E2 10740.86} C_VEL
LIN {X 0,Y 558.651,Z 1074.06,A -85,B 0,C 180,E1 10745.162,E2 10745.162} C_VEL
LIN {X 0,Y 566.191,Z 1035.379,A -85,B 0,C 180,E1 10748.823,E2 10748.823} C_VEL
LIN {X 0,Y 574.37,Z 991.637,A -85,B 0,C 180,E1 10752.029,E2 10752.029} C_VEL
LIN {X 0,Y 581.413,Z 949.818,A -85,B 0,C 180,E1 10754.39,E2 10754.39} C_VEL
LIN {X 0,Y 587.822,Z 901.976,A -85,B 0,C 180,E1 10756.391,E2 10756.391} C_VEL
LIN {X 0,Y 592.36,Z 852.414,A -85,B 0,C 180,E1 10757.849,E2 10757.849} C_VEL
LIN {X 0,Y 571.682,Z 814.77,A -85,B 0,C 180,E1 10761.169,E2 10761.169} C_VEL
LIN {X 0,Y 549.351,Z 780.853,A -85,B 0,C 180,E1 10764.889,E2 10764.889} C_VEL
LIN {X 0,Y 540.156,Z 768.018,A -85,B 0,C 180,E1 10766.591,E2 10766.591} C_VEL
LIN {X 0,Y 537.5,Z 763.206,A -85,B 0,C 180,E1 10767.134,E2 10767.134} C_VEL
LIN {X 0,Y 537.422,Z 762.06,A -85,B 0,C 180,E1 10767.352,E2 10767.352} C_VEL
LIN {X 0,Y 537.621,Z 762.06,A -85,B 0,C 180,E1 10773.268,E2 10773.268} C_VEL
LIN {X 0,Y 537.733,Z 762.06,A -85,B 0,C 180,E1 10778.566,E2 10778.566} C_VEL
LIN {X 0,Y 537.948,Z 762.06,A -85,B 0,C 180,E1 10783.678,E2 10783.678} C_VEL
LIN {X 0,Y 538.17,Z 762.06,A -85,B 0,C 180,E1 10789.339,E2 10789.339} C_VEL
LIN {X 0,Y 538.471,Z 762.06,A -85,B 0,C 180,E1 10795.162,E2 10795.162} C_VEL
LIN {X 0,Y 538.705,Z 762.06,A -85,B 0,C 180,E1 10799.991,E2 10799.991} C_VEL
LIN {X 0,Y 538.482,Z 762.06,A -85,B 0,C 180,E1 10804.819,E2 10804.819} C_VEL
LIN {X 0,Y 538.117,Z 762.06,A -85,B 0,C 180,E1 10810.631,E2 10810.631} C_VEL
LIN {X 0,Y 537.742,Z 762.06,A -85,B 0,C 180,E1 10816.309,E2 10816.309} C_VEL
LIN {X 0,Y 537.639,Z 762.06,A -85,B 0,C 180,E1 10821.952,E2 10821.952} C_VEL
LIN {X 0,Y 537.633,Z 762.06,A -85,B 0,C 180,E1 10826.711,E2 10826.711} C_VEL
LIN {X 0,Y 537.448,Z 762.06,A -85,B 0,C 180,E1 10832.871,E2 10832.871} C_VEL
LIN {X 0,Y 537.47,Z 762.235,A -85,B 0,C 180,E1 10833.255,E2 10833.255} C_VEL
LIN {X 0,Y 539.778,Z 767.583,A -85,B 0,C 180,E1 10833.756,E2 10833.756} C_VEL
LIN {X 0,Y 542.693,Z 771.454,A -85,B 0,C 180,E1 10834.307,E2 10834.307} C_VEL
LIN {X 0,Y 562.138,Z 799.96,A -85,B 0,C 180,E1 10837.761,E2 10837.761} C_VEL
LIN {X 0,Y 582.23,Z 835.465,A -85,B 0,C 180,E1 10841.295,E2 10841.295} C_VEL
LIN {X 0,Y 590.723,Z 854.183,A -85,B 0,C 180,E1 10842.934,E2 10842.934} C_VEL
LIN {X 0,Y 584.706,Z 901.813,A -85,B 0,C 180,E1 10844.628,E2 10844.628} C_VEL
LIN {X 0,Y 577.585,Z 946.939,A -85,B 0,C 180,E1 10846.918,E2 10846.918} C_VEL
LIN {X 0,Y 569.493,Z 990.854,A -85,B 0,C 180,E1 10849.882,E2 10849.882} C_VEL
LIN {X 0,Y 561.65,Z 1029.694,A -85,B 0,C 180,E1 10853.3,E2 10853.3} C_VEL
LIN {X 0,Y 554.134,Z 1067.094,A -85,B 0,C 180,E1 10857.457,E2 10857.457} C_VEL
LIN {X 0,Y 547.951,Z 1099.399,A -85,B 0,C 180,E1 10862.043,E2 10862.043} C_VEL
LIN {X 0,Y 543.698,Z 1125.589,A -85,B 0,C 180,E1 10866.752,E2 10866.752} C_VEL
LIN {X 0,Y 540.938,Z 1146.746,A -85,B 0,C 180,E1 10871.715,E2 10871.715} C_VEL
LIN {X 0,Y 539.452,Z 1162.425,A -85,B 0,C 180,E1 10876.639,E2 10876.639} C_VEL
LIN {X 0,Y 538.837,Z 1172.305,A -85,B 0,C 180,E1 10881.128,E2 10881.128} C_VEL
LIN {X 0,Y 538.55,Z 1177.706,A -85,B 0,C 180,E1 10885.172,E2 10885.172} C_VEL
LIN {X 0,Y 538.619,Z 1179.997,A -85,B 0,C 180,E1 10890.001,E2 10890.001} C_VEL
LIN {X 0,Y 538.64,Z 1177.608,A -85,B 0,C 180,E1 10894.829,E2 10894.829} C_VEL
LIN {X 0,Y 538.892,Z 1170.58,A -85,B 0,C 180,E1 10899.687,E2 10899.687} C_VEL
LIN {X 0,Y 539.7,Z 1158.734,A -85,B 0,C 180,E1 10904.596,E2 10904.596} C_VEL
LIN {X 0,Y 541.453,Z 1141.508,A -85,B 0,C 180,E1 10909.567,E2 10909.567} C_VEL
LIN {X 0,Y 544.832,Z 1118.262,A -85,B 0,C 180,E1 10914.585,E2 10914.585} C_VEL
LIN {X 0,Y 549.623,Z 1090.614,A -85,B 0,C 180,E1 10919.229,E2 10919.229} C_VEL
LIN {X 0,Y 556.517,Z 1054.97,A -85,B 0,C 180,E1 10923.908,E2 10923.908} C_VEL
LIN {X 0,Y 564.385,Z 1016.162,A -85,B 0,C 180,E1 10927.895,E2 10927.895} C_VEL
LIN {X 0,Y 572.366,Z 975.736,A -85,B 0,C 180,E1 10931.153,E2 10931.153} C_VEL
LIN {X 0,Y 580.462,Z 930.141,A -85,B 0,C 180,E1 10933.917,E2 10933.917} C_VEL
LIN {X 0,Y 586.813,Z 887.807,A -85,B 0,C 180,E1 10935.838,E2 10935.838} C_VEL
LIN {X 0,Y 590.165,Z 852.289,A -85,B 0,C 180,E1 10937.114,E2 10937.114} C_VEL
LIN {X 0,Y 573.034,Z 818.153,A -85,B 0,C 180,E1 10940.26,E2 10940.26} C_VEL
LIN {X 0,Y 550.118,Z 781.628,A -85,B 0,C 180,E1 10944.244,E2 10944.244} C_VEL
LIN {X 0,Y 540.243,Z 768.079,A -85,B 0,C 180,E1 10946.056,E2 10946.056} C_VEL
LIN {X 0,Y 537.57,Z 763.576,A -85,B 0,C 180,E1 10946.594,E2 10946.594} C_VEL
LIN {X 0,Y 537.422,Z 762.06,A -85,B 0,C 180,E1 10946.695,E2 10946.695} C_VEL
LIN {X 0,Y 537.473,Z 762.06,A -85,B 0,C 180,E1 10951.463,E2 10951.463} C_VEL
LIN {X 0,Y 537.582,Z 762.06,A -85,B 0,C 180,E1 10956.839,E2 10956.839} C_VEL
LIN {X 0,Y 537.712,Z 762.06,A -85,B 0,C 180,E1 10962.843,E2 10962.843} C_VEL
LIN {X 0,Y 538.124,Z 762.06,A -85,B 0,C 180,E1 10968.675,E2 10968.675} C_VEL
LIN {X 0,Y 538.366,Z 762.06,A -85,B 0,C 180,E1 10973.564,E2 10973.564} C_VEL
LIN {X 0,Y 538.561,Z 762.06,A -85,B 0,C 180,E1 10978.402,E2 10978.402} C_VEL
LIN {X 0,Y 538.459,Z 762.06,A -85,B 0,C 180,E1 10983.226,E2 10983.226} C_VEL
LIN {X 0,Y 538.286,Z 762.06,A -85,B 0,C 180,E1 10988.077,E2 10988.077} C_VEL
LIN {X 0,Y 538.105,Z 762.06,A -85,B 0,C 180,E1 10992.991,E2 10992.991} C_VEL
LIN {X 0,Y 537.983,Z 762.06,A -85,B 0,C 180,E1 10998.005,E2 10998.005} C_VEL
LIN {X 0,Y 537.808,Z 762.06,A -85,B 0,C 180,E1 11003.171,E2 11003.171} C_VEL
LIN {X 0,Y 537.678,Z 762.06,A -85,B 0,C 180,E1 11008.547,E2 11008.547} C_VEL
LIN {X 0,Y 537.506,Z 762.06,A -85,B 0,C 180,E1 11012.827,E2 11012.827} C_VEL
LIN {X 0,Y 539.704,Z 767.513,A -85,B 0,C 180,E1 11013.338,E2 11013.338} C_VEL
LIN {X 0,Y 542.506,Z 770.969,A -85,B 0,C 180,E1 11013.861,E2 11013.861} C_VEL
LIN {X 0,Y 564.042,Z 802.782,A -85,B 0,C 180,E1 11017.619,E2 11017.619} C_VEL
LIN {X 0,Y 585.129,Z 838.228,A -85,B 0,C 180,E1 11020.971,E2 11020.971} C_VEL
LIN {X 0,Y 592.977,Z 854.349,A -85,B 0,C 180,E1 11022.273,E2 11022.273} C_VEL
LIN {X 0,Y 587.596,Z 903.829,A -85,B 0,C 180,E1 11023.674,E2 11023.674} C_VEL
LIN {X 0,Y 581.588,Z 948.41,A -85,B 0,C 180,E1 11025.541,E2 11025.541} C_VEL
LIN {X 0,Y 574.31,Z 991.752,A -85,B 0,C 180,E1 11027.976,E2 11027.976} C_VEL
LIN {X 0,Y 566.158,Z 1035.464,A -85,B 0,C 180,E1 11031.183,E2 11031.183} C_VEL
LIN {X 0,Y 558.668,Z 1074.033,A -85,B 0,C 180,E1 11034.836,E2 11034.836} C_VEL
LIN {X 0,Y 557.762,Z 1078.73,A -85,B 0,C 180,E1 11035.351,E2 11035.351} C_VEL
LIN {X 0,Y 551.944,Z 1090.849,A -85,B 0,C 180,E1 11036.512,E2 11036.512} C_VEL
LIN {X 0,Y 546.03,Z 1102.423,A -85,B 0,C 180,E1 11037.741,E2 11037.741} C_VEL
LIN {X 0,Y 539.789,Z 1134.402,A -85,B 0,C 180,E1 11042.489,E2 11042.489} C_VEL
LIN {X 0,Y 535.276,Z 1160.867,A -85,B 0,C 180,E1 11047.597,E2 11047.597} C_VEL
LIN {X 0,Y 532.694,Z 1181.016,A -85,B 0,C 180,E1 11052.67,E2 11052.67} C_VEL
LIN {X 0,Y 531.333,Z 1195.38,A -85,B 0,C 180,E1 11057.683,E2 11057.683} C_VEL
LIN {X 0,Y 530.868,Z 1204.744,A -85,B 0,C 180,E1 11062.64,E2 11062.64} C_VEL
LIN {X 0,Y 530.761,Z 1208.898,A -85,B 0,C 180,E1 11066.735,E2 11066.735} C_VEL
LIN {X 0,Y 530.96,Z 1209.666,A -85,B 0,C 180,E1 11071.63,E2 11071.63} C_VEL
LIN {X 0,Y 530.879,Z 1205.911,A -85,B 0,C 180,E1 11076.537,E2 11076.537} C_VEL
LIN {X 0,Y 531.223,Z 1197.305,A -85,B 0,C 180,E1 11081.485,E2 11081.485} C_VEL
LIN {X 0,Y 532.324,Z 1183.705,A -85,B 0,C 180,E1 11086.49,E2 11086.49} C_VEL
LIN {X 0,Y 534.719,Z 1164.741,A -85,B 0,C 180,E1 11091.553,E2 11091.553} C_VEL
LIN {X 0,Y 538.895,Z 1139.227,A -85,B 0,C 180,E1 11096.656,E2 11096.656} C_VEL
LIN {X 0,Y 544.767,Z 1108.857,A -85,B 0,C 180,E1 11101.4,E2 11101.4} C_VEL
LIN {X 0,Y 551.732,Z 1074.38,A -85,B 0,C 180,E1 11105.597,E2 11105.597} C_VEL
LIN {X 0,Y 559.342,Z 1037.287,A -85,B 0,C 180,E1 11109.175,E2 11109.175} C_VEL
LIN {X 0,Y 567.565,Z 995.323,A -85,B 0,C 180,E1 11112.321,E2 11112.321} C_VEL
LIN {X 0,Y 575.131,Z 952.476,A -85,B 0,C 180,E1 11114.809,E2 11114.809} C_VEL
LIN {X 0,Y 581.735,Z 906.059,A -85,B 0,C 180,E1 11116.813,E2 11116.813} C_VEL
LIN {X 0,Y 586.767,Z 855.846,A -85,B 0,C 180,E1 11118.336,E2 11118.336} C_VEL
LIN {X 0,Y 566.856,Z 819.189,A -85,B 0,C 180,E1 11121.669,E2 11121.669} C_VEL
LIN {X 0,Y 545.755,Z 786.891,A -85,B 0,C 180,E1 11125.289,E2 11125.289} C_VEL
LIN {X 0,Y 532.404,Z 768.173,A -85,B 0,C 180,E1 11127.863,E2 11127.863} C_VEL
LIN {X 0,Y 529.626,Z 763.533,A -85,B 0,C 180,E1 11128.457,E2 11128.457} C_VEL
LIN {X 0,Y 529.487,Z 762.06,A -85,B 0,C 180,E1 11128.726,E2 11128.726} C_VEL
LIN {X 0,Y 529.702,Z 762.06,A -85,B 0,C 180,E1 11134.658,E2 11134.658} C_VEL
LIN {X 0,Y 529.943,Z 762.06,A -85,B 0,C 180,E1 11140.215,E2 11140.215} C_VEL
LIN {X 0,Y 530.104,Z 762.06,A -85,B 0,C 180,E1 11145.74,E2 11145.74} C_VEL
LIN {X 0,Y 530.353,Z 762.06,A -85,B 0,C 180,E1 11151.801,E2 11151.801} C_VEL
LIN {X 0,Y 530.544,Z 762.06,A -85,B 0,C 180,E1 11156.725,E2 11156.725} C_VEL
LIN {X 0,Y 530.648,Z 762.06,A -85,B 0,C 180,E1 11161.622,E2 11161.622} C_VEL
LIN {X 0,Y 530.489,Z 762.06,A -85,B 0,C 180,E1 11166.532,E2 11166.532} C_VEL
LIN {X 0,Y 530.177,Z 762.06,A -85,B 0,C 180,E1 11171.497,E2 11171.497} C_VEL
LIN {X 0,Y 529.82,Z 762.06,A -85,B 0,C 180,E1 11176.559,E2 11176.559} C_VEL
LIN {X 0,Y 529.758,Z 762.06,A -85,B 0,C 180,E1 11181.753,E2 11181.753} C_VEL
LIN {X 0,Y 529.652,Z 762.06,A -85,B 0,C 180,E1 11187.819,E2 11187.819} C_VEL
LIN {X 0,Y 529.585,Z 762.708,A -85,B 0,C 180,E1 11191.931,E2 11191.931} C_VEL
LIN {X 0,Y 532.232,Z 767.986,A -85,B 0,C 180,E1 11192.52,E2 11192.52} C_VEL
LIN {X 0,Y 535.093,Z 771.878,A -85,B 0,C 180,E1 11193.096,E2 11193.096} C_VEL
LIN {X 0,Y 551.943,Z 796.049,A -85,B 0,C 180,E1 11196.259,E2 11196.259} C_VEL
LIN {X 0,Y 571.264,Z 828.583,A -85,B 0,C 180,E1 11199.749,E2 11199.749} C_VEL
LIN {X 0,Y 584.974,Z 857.686,A -85,B 0,C 180,E1 11202.462,E2 11202.462} C_VEL
LIN {X 0,Y 578.796,Z 904.333,A -85,B 0,C 180,E1 11204.159,E2 11204.159} C_VEL
LIN {X 0,Y 571.187,Z 950.113,A -85,B 0,C 180,E1 11206.541,E2 11206.541} C_VEL
LIN {X 0,Y 562.811,Z 993.612,A -85,B 0,C 180,E1 11209.543,E2 11209.543} C_VEL
LIN {X 0,Y 554.376,Z 1033.478,A -85,B 0,C 180,E1 11213.155,E2 11213.155} C_VEL
LIN {X 0,Y 546.657,Z 1069.453,A -85,B 0,C 180,E1 11217.301,E2 11217.301} C_VEL
LIN {X 0,Y 540.153,Z 1102.04,A -85,B 0,C 180,E1 11222.058,E2 11222.058} C_VEL
LIN {X 0,Y 535.869,Z 1127.178,A -85,B 0,C 180,E1 11226.748,E2 11226.748} C_VEL
LIN {X 0,Y 532.866,Z 1149.691,A -85,B 0,C 180,E1 11232.252,E2 11232.252} C_VEL
LIN {X 0,Y 531.487,Z 1163.534,A -85,B 0,C 180,E1 11236.854,E2 11236.854} C_VEL
LIN {X 0,Y 530.92,Z 1173.606,A -85,B 0,C 180,E1 11241.819,E2 11241.819} C_VEL
LIN {X 0,Y 530.673,Z 1178.928,A -85,B 0,C 180,E1 11246.736,E2 11246.736} C_VEL
LIN {X 0,Y 530.795,Z 1179.656,A -85,B 0,C 180,E1 11251.632,E2 11251.632} C_VEL
LIN {X 0,Y 530.905,Z 1175.853,A -85,B 0,C 180,E1 11256.538,E2 11256.538} C_VEL
LIN {X 0,Y 531.246,Z 1167.198,A -85,B 0,C 180,E1 11261.486,E2 11261.486} C_VEL
LIN {X 0,Y 532.579,Z 1152.222,A -85,B 0,C 180,E1 11266.908,E2 11266.908} C_VEL
LIN {X 0,Y 535.048,Z 1132.611,A -85,B 0,C 180,E1 11271.977,E2 11271.977} C_VEL
LIN {X 0,Y 539.325,Z 1106.581,A -85,B 0,C 180,E1 11277.085,E2 11277.085} C_VEL
LIN {X 0,Y 545.09,Z 1077.084,A -85,B 0,C 180,E1 11281.593,E2 11281.593} C_VEL
LIN {X 0,Y 552.885,Z 1040.237,A -85,B 0,C 180,E1 11286.066,E2 11286.066} C_VEL
LIN {X 0,Y 561.263,Z 1001.168,A -85,B 0,C 180,E1 11289.735,E2 11289.735} C_VEL
LIN {X 0,Y 569.325,Z 960.889,A -85,B 0,C 180,E1 11292.697,E2 11292.697} C_VEL
LIN {X 0,Y 576.961,Z 915.775,A -85,B 0,C 180,E1 11295.22,E2 11295.22} C_VEL
LIN {X 0,Y 583.83,Z 867.088,A -85,B 0,C 180,E1 11297.174,E2 11297.174} C_VEL
LIN {X 0,Y 584.412,Z 855.585,A -85,B 0,C 180,E1 11297.597,E2 11297.597} C_VEL
LIN {X 0,Y 567.227,Z 821.031,A -85,B 0,C 180,E1 11300.891,E2 11300.891} C_VEL
LIN {X 0,Y 546.509,Z 787.713,A -85,B 0,C 180,E1 11304.641,E2 11304.641} C_VEL
LIN {X 0,Y 532.646,Z 768.348,A -85,B 0,C 180,E1 11307.296,E2 11307.296} C_VEL
LIN {X 0,Y 529.677,Z 763.772,A -85,B 0,C 180,E1 11307.92,E2 11307.92} C_VEL
LIN {X 0,Y 529.496,Z 762.06,A -85,B 0,C 180,E1 11308.075,E2 11308.075} C_VEL
LIN {X 0,Y 529.571,Z 762.06,A -85,B 0,C 180,E1 11312.849,E2 11312.849} C_VEL
LIN {X 0,Y 529.688,Z 762.06,A -85,B 0,C 180,E1 11318.244,E2 11318.244} C_VEL
LIN {X 0,Y 529.827,Z 762.06,A -85,B 0,C 180,E1 11323.441,E2 11323.441} C_VEL
LIN {X 0,Y 530.192,Z 762.06,A -85,B 0,C 180,E1 11328.503,E2 11328.503} C_VEL
LIN {X 0,Y 530.466,Z 762.06,A -85,B 0,C 180,E1 11333.468,E2 11333.468} C_VEL
LIN {X 0,Y 530.658,Z 762.06,A -85,B 0,C 180,E1 11338.378,E2 11338.378} C_VEL
LIN {X 0,Y 530.553,Z 762.06,A -85,B 0,C 180,E1 11343.275,E2 11343.275} C_VEL
LIN {X 0,Y 530.367,Z 762.06,A -85,B 0,C 180,E1 11348.199,E2 11348.199} C_VEL
LIN {X 0,Y 530.135,Z 762.06,A -85,B 0,C 180,E1 11354.267,E2 11354.267} C_VEL
LIN {X 0,Y 530.036,Z 762.06,A -85,B 0,C 180,E1 11360.013,E2 11360.013} C_VEL
LIN {X 0,Y 529.819,Z 762.06,A -85,B 0,C 180,E1 11365.336,E2 11365.336} C_VEL
LIN {X 0,Y 529.624,Z 762.06,A -85,B 0,C 180,E1 11371.508,E2 11371.508} C_VEL
LIN {X 0,Y 531.546,Z 767.241,A -85,B 0,C 180,E1 11371.983,E2 11371.983} C_VEL
LIN {X 0,Y 534.635,Z 770.902,A -85,B 0,C 180,E1 11372.593,E2 11372.593} C_VEL
LIN {X 0,Y 555.12,Z 800.506,A -85,B 0,C 180,E1 11376.37,E2 11376.37} C_VEL
LIN {X 0,Y 577.406,Z 837.441,A -85,B 0,C 180,E1 11380.069,E2 11380.069} C_VEL
LIN {X 0,Y 587.221,Z 858.257,A -85,B 0,C 180,E1 11381.797,E2 11381.797} C_VEL
LIN {X 0,Y 581.768,Z 905.951,A -85,B 0,C 180,E1 11383.185,E2 11383.185} C_VEL
LIN {X 0,Y 575.362,Z 951.041,A -85,B 0,C 180,E1 11385.114,E2 11385.114} C_VEL
LIN {X 0,Y 567.531,Z 995.35,A -85,B 0,C 180,E1 11387.679,E2 11387.679} C_VEL
LIN {X 0,Y 559.316,Z 1037.354,A -85,B 0,C 180,E1 11390.83,E2 11390.83} C_VEL
LIN {X 0,Y 551.211,Z 1076.981,A -85,B 0,C 180,E1 11394.687,E2 11394.687} C_VEL
LIN {X 0,Y 546.03,Z 1102.423,A -85,B 0,C 180,E1 11397.741,E2 11397.741} C_VEL
LIN {X 0,Y 540.129,Z 1113.589,A -85,B 0,C 180,E1 11399.03,E2 11399.03} C_VEL
LIN {X 0,Y 534.439,Z 1124.124,A -85,B 0,C 180,E1 11400.395,E2 11400.395} C_VEL
LIN {X 0,Y 529.056,Z 1152.626,A -85,B 0,C 180,E1 11405.494,E2 11405.494} C_VEL
LIN {X 0,Y 525.852,Z 1173.389,A -85,B 0,C 180,E1 11410.265,E2 11410.265} C_VEL
LIN {X 0,Y 523.994,Z 1189.998,A -85,B 0,C 180,E1 11415.383,E2 11415.383} C_VEL
LIN {X 0,Y 523.148,Z 1200.66,A -85,B 0,C 180,E1 11420.019,E2 11420.019} C_VEL
LIN {X 0,Y 522.826,Z 1207.65,A -85,B 0,C 180,E1 11425.025,E2 11425.025} C_VEL
LIN {X 0,Y 522.936,Z 1210,A -85,B 0,C 180,E1 11429.999,E2 11429.999} C_VEL
LIN {X 0,Y 522.826,Z 1207.653,A -85,B 0,C 180,E1 11434.973,E2 11434.973} C_VEL
LIN {X 0,Y 523.138,Z 1200.664,A -85,B 0,C 180,E1 11439.98,E2 11439.98} C_VEL
LIN {X 0,Y 524.162,Z 1188.258,A -85,B 0,C 180,E1 11445.262,E2 11445.262} C_VEL
LIN {X 0,Y 526.203,Z 1170.574,A -85,B 0,C 180,E1 11450.44,E2 11450.44} C_VEL
LIN {X 0,Y 529.891,Z 1147.28,A -85,B 0,C 180,E1 11455.576,E2 11455.576} C_VEL
LIN {X 0,Y 535.385,Z 1119.571,A -85,B 0,C 180,E1 11460.298,E2 11460.298} C_VEL
LIN {X 0,Y 542.447,Z 1086.021,A -85,B 0,C 180,E1 11464.763,E2 11464.763} C_VEL
LIN {X 0,Y 550.415,Z 1048.994,A -85,B 0,C 180,E1 11468.632,E2 11468.632} C_VEL
LIN {X 0,Y 559.263,Z 1006.434,A -85,B 0,C 180,E1 11472.11,E2 11472.11} C_VEL
LIN {X 0,Y 567.218,Z 964.182,A -85,B 0,C 180,E1 11474.761,E2 11474.761} C_VEL
LIN {X 0,Y 574.939,Z 915.36,A -85,B 0,C 180,E1 11477.044,E2 11477.044} C_VEL
LIN {X 0,Y 580.738,Z 868.226,A -85,B 0,C 180,E1 11478.558,E2 11478.558} C_VEL
LIN {X 0,Y 581.028,Z 858.987,A -85,B 0,C 180,E1 11478.854,E2 11478.854} C_VEL
LIN {X 0,Y 560.909,Z 821.603,A -85,B 0,C 180,E1 11482.378,E2 11482.378} C_VEL
LIN {X 0,Y 538.968,Z 788.033,A -85,B 0,C 180,E1 11486.31,E2 11486.31} C_VEL
LIN {X 0,Y 524.63,Z 768.252,A -85,B 0,C 180,E1 11489.227,E2 11489.227} C_VEL
LIN {X 0,Y 521.683,Z 763.29,A -85,B 0,C 180,E1 11489.903,E2 11489.903} C_VEL
LIN {X 0,Y 521.585,Z 762.06,A -85,B 0,C 180,E1 11489.954,E2 11489.954} C_VEL
LIN {X 0,Y 521.791,Z 762.06,A -85,B 0,C 180,E1 11496.074,E2 11496.074} C_VEL
LIN {X 0,Y 522.019,Z 762.06,A -85,B 0,C 180,E1 11501.425,E2 11501.425} C_VEL
LIN {X 0,Y 522.237,Z 762.06,A -85,B 0,C 180,E1 11506.607,E2 11506.607} C_VEL
LIN {X 0,Y 522.435,Z 762.06,A -85,B 0,C 180,E1 11511.676,E2 11511.676} C_VEL
LIN {X 0,Y 522.641,Z 762.06,A -85,B 0,C 180,E1 11516.676,E2 11516.676} C_VEL
LIN {X 0,Y 522.763,Z 762.06,A -85,B 0,C 180,E1 11521.647,E2 11521.647} C_VEL
LIN {X 0,Y 522.571,Z 762.06,A -85,B 0,C 180,E1 11526.632,E2 11526.632} C_VEL
LIN {X 0,Y 522.268,Z 762.06,A -85,B 0,C 180,E1 11531.674,E2 11531.674} C_VEL
LIN {X 0,Y 521.863,Z 762.06,A -85,B 0,C 180,E1 11537.15,E2 11537.15} C_VEL
LIN {X 0,Y 521.822,Z 762.06,A -85,B 0,C 180,E1 11542.101,E2 11542.101} C_VEL
LIN {X 0,Y 521.779,Z 762.06,A -85,B 0,C 180,E1 11547.59,E2 11547.59} C_VEL
LIN {X 0,Y 521.686,Z 762.612,A -85,B 0,C 180,E1 11550.496,E2 11550.496} C_VEL
LIN {X 0,Y 524.091,Z 767.757,A -85,B 0,C 180,E1 11551.078,E2 11551.078} C_VEL
LIN {X 0,Y 526.676,Z 770.659,A -85,B 0,C 180,E1 11551.62,E2 11551.62} C_VEL
LIN {X 0,Y 547.793,Z 801.181,A -85,B 0,C 180,E1 11555.793,E2 11555.793} C_VEL
LIN {X 0,Y 567.849,Z 836.066,A -85,B 0,C 180,E1 11559.611,E2 11559.611} C_VEL
LIN {X 0,Y 579.313,Z 861.1,A -85,B 0,C 180,E1 11561.983,E2 11561.983} C_VEL
LIN {X 0,Y 572.842,Z 907.145,A -85,B 0,C 180,E1 11563.702,E2 11563.702} C_VEL
LIN {X 0,Y 564.444,Z 955.175,A -85,B 0,C 180,E1 11566.269,E2 11566.269} C_VEL
LIN {X 0,Y 556.312,Z 995.31,A -85,B 0,C 180,E1 11569.119,E2 11569.119} C_VEL
LIN {X 0,Y 547.386,Z 1035.823,A -85,B 0,C 180,E1 11572.854,E2 11572.854} C_VEL
LIN {X 0,Y 539.647,Z 1069.96,A -85,B 0,C 180,E1 11576.873,E2 11576.873} C_VEL
LIN {X 0,Y 532.618,Z 1103.236,A -85,B 0,C 180,E1 11581.837,E2 11581.837} C_VEL
LIN {X 0,Y 527.987,Z 1129.119,A -85,B 0,C 180,E1 11586.827,E2 11586.827} C_VEL
LIN {X 0,Y 525.076,Z 1149.919,A -85,B 0,C 180,E1 11592.045,E2 11592.045} C_VEL
LIN {X 0,Y 523.655,Z 1163.532,A -85,B 0,C 180,E1 11596.653,E2 11596.653} C_VEL
LIN {X 0,Y 523.024,Z 1173.602,A -85,B 0,C 180,E1 11601.695,E2 11601.695} C_VEL
LIN {X 0,Y 522.779,Z 1178.925,A -85,B 0,C 180,E1 11606.687,E2 11606.687} C_VEL
LIN {X 0,Y 522.895,Z 1179.656,A -85,B 0,C 180,E1 11611.657,E2 11611.657} C_VEL
LIN {X 0,Y 523.003,Z 1175.854,A -85,B 0,C 180,E1 11616.637,E2 11616.637} C_VEL
LIN {X 0,Y 523.401,Z 1167.196,A -85,B 0,C 180,E1 11621.66,E2 11621.66} C_VEL
LIN {X 0,Y 524.796,Z 1152.307,A -85,B 0,C 180,E1 11627.14,E2 11627.14} C_VEL
LIN {X 0,Y 527.385,Z 1132.613,A -85,B 0,C 180,E1 11632.313,E2 11632.313} C_VEL
LIN {X 0,Y 532.116,Z 1105.858,A -85,B 0,C 180,E1 11637.622,E2 11637.622} C_VEL
LIN {X 0,Y 538.659,Z 1074.265,A -85,B 0,C 180,E1 11642.45,E2 11642.45} C_VEL
LIN {X 0,Y 546.682,Z 1038.912,A -85,B 0,C 180,E1 11646.742,E2 11646.742} C_VEL
LIN {X 0,Y 555.266,Z 1000.175,A -85,B 0,C 180,E1 11650.382,E2 11650.382} C_VEL
LIN {X 0,Y 563.579,Z 960.148,A -85,B 0,C 180,E1 11653.327,E2 11653.327} C_VEL
LIN {X 0,Y 571.735,Z 913.929,A -85,B 0,C 180,E1 11655.886,E2 11655.886} C_VEL
LIN {X 0,Y 578.519,Z 866.926,A -85,B 0,C 180,E1 11657.764,E2 11657.764} C_VEL
LIN {X 0,Y 578.754,Z 859.103,A -85,B 0,C 180,E1 11658.075,E2 11658.075} C_VEL
LIN {X 0,Y 562.057,Z 825.061,A -85,B 0,C 180,E1 11661.425,E2 11661.425} C_VEL
LIN {X 0,Y 542.499,Z 793.325,A -85,B 0,C 180,E1 11665.11,E2 11665.11} C_VEL
LIN {X 0,Y 528.398,Z 773.71,A -85,B 0,C 180,E1 11667.892,E2 11667.892} C_VEL
LIN {X 0,Y 524.899,Z 768.509,A -85,B 0,C 180,E1 11668.647,E2 11668.647} C_VEL
LIN {X 0,Y 521.756,Z 763.823,A -85,B 0,C 180,E1 11669.349,E2 11669.349} C_VEL
LIN {X 0,Y 521.575,Z 762.06,A -85,B 0,C 180,E1 11669.51,E2 11669.51} C_VEL
LIN {X 0,Y 521.664,Z 762.06,A -85,B 0,C 180,E1 11674.26,E2 11674.26} C_VEL
LIN {X 0,Y 521.755,Z 762.06,A -85,B 0,C 180,E1 11679.676,E2 11679.676} C_VEL
LIN {X 0,Y 522.006,Z 762.06,A -85,B 0,C 180,E1 11684.91,E2 11684.91} C_VEL
LIN {X 0,Y 522.395,Z 762.06,A -85,B 0,C 180,E1 11690.016,E2 11690.016} C_VEL
LIN {X 0,Y 522.64,Z 762.06,A -85,B 0,C 180,E1 11695.034,E2 11695.034} C_VEL
LIN {X 0,Y 522.926,Z 762.06,A -85,B 0,C 180,E1 11700.01,E2 11700.01} C_VEL
LIN {X 0,Y 522.545,Z 762.06,A -85,B 0,C 180,E1 11706.651,E2 11706.651} C_VEL
LIN {X 0,Y 522.334,Z 762.06,A -85,B 0,C 180,E1 11711.692,E2 11711.692} C_VEL
LIN {X 0,Y 522.127,Z 762.06,A -85,B 0,C 180,E1 11717.238,E2 11717.238} C_VEL
LIN {X 0,Y 521.998,Z 762.06,A -85,B 0,C 180,E1 11722.124,E2 11722.124} C_VEL
LIN {X 0,Y 521.881,Z 762.06,A -85,B 0,C 180,E1 11727.606,E2 11727.606} C_VEL
LIN {X 0,Y 521.76,Z 762.676,A -85,B 0,C 180,E1 11730.115,E2 11730.115} C_VEL
LIN {X 0,Y 524.182,Z 767.754,A -85,B 0,C 180,E1 11730.696,E2 11730.696} C_VEL
LIN {X 0,Y 526.858,Z 770.978,A -85,B 0,C 180,E1 11731.261,E2 11731.261} C_VEL
LIN {X 0,Y 546.158,Z 798.628,A -85,B 0,C 180,E1 11735.044,E2 11735.044} C_VEL
LIN {X 0,Y 567.898,Z 833.474,A -85,B 0,C 180,E1 11738.809,E2 11738.809} C_VEL
LIN {X 0,Y 581.614,Z 861.077,A -85,B 0,C 180,E1 11741.286,E2 11741.286} C_VEL
LIN {X 0,Y 576.099,Z 907.285,A -85,B 0,C 180,E1 11742.66,E2 11742.66} C_VEL
LIN {X 0,Y 569.545,Z 951.373,A -85,B 0,C 180,E1 11744.571,E2 11744.571} C_VEL
LIN {X 0,Y 561.195,Z 996.592,A -85,B 0,C 180,E1 11747.215,E2 11747.215} C_VEL
LIN {X 0,Y 552.715,Z 1037.953,A -85,B 0,C 180,E1 11750.364,E2 11750.364} C_VEL
LIN {X 0,Y 544.167,Z 1078.026,A -85,B 0,C 180,E1 11754.326,E2 11754.326} C_VEL
LIN {X 0,Y 537.287,Z 1110.825,A -85,B 0,C 180,E1 11758.41,E2 11758.41} C_VEL
LIN {X 0,Y 534.439,Z 1124.124,A -85,B 0,C 180,E1 11760.395,E2 11760.395} C_VEL
LIN {X 0,Y 528.875,Z 1134.212,A -85,B 0,C 180,E1 11761.836,E2 11761.836} C_VEL
LIN {X 0,Y 523.303,Z 1143.56,A -85,B 0,C 180,E1 11763.323,E2 11763.323} C_VEL
LIN {X 0,Y 519.108,Z 1166.935,A -85,B 0,C 180,E1 11768.328,E2 11768.328} C_VEL
LIN {X 0,Y 516.62,Z 1185.03,A -85,B 0,C 180,E1 11773.429,E2 11773.429} C_VEL
LIN {X 0,Y 515.483,Z 1197.296,A -85,B 0,C 180,E1 11778.158,E2 11778.158} C_VEL
LIN {X 0,Y 515.091,Z 1205.908,A -85,B 0,C 180,E1 11783.26,E2 11783.26} C_VEL
LIN {X 0,Y 514.889,Z 1209.666,A -85,B 0,C 180,E1 11788.317,E2 11788.317} C_VEL
LIN {X 0,Y 515.151,Z 1209.666,A -85,B 0,C 180,E1 11791.68,E2 11791.68} C_VEL
LIN {X 0,Y 515.098,Z 1205.911,A -85,B 0,C 180,E1 11796.738,E2 11796.738} C_VEL
LIN {X 0,Y 515.479,Z 1197.299,A -85,B 0,C 180,E1 11801.841,E2 11801.841} C_VEL
LIN {X 0,Y 516.764,Z 1183.704,A -85,B 0,C 180,E1 11807.002,E2 11807.002} C_VEL
LIN {X 0,Y 519.49,Z 1164.742,A -85,B 0,C 180,E1 11812.218,E2 11812.218} C_VEL
LIN {X 0,Y 524.125,Z 1139.222,A -85,B 0,C 180,E1 11817.47,E2 11817.47} C_VEL
LIN {X 0,Y 530.224,Z 1110.6,A -85,B 0,C 180,E1 11822.059,E2 11822.059} C_VEL
LIN {X 0,Y 538.203,Z 1074.16,A -85,B 0,C 180,E1 11826.592,E2 11826.592} C_VEL
LIN {X 0,Y 546.788,Z 1035.848,A -85,B 0,C 180,E1 11830.347,E2 11830.347} C_VEL
LIN {X 0,Y 556.009,Z 992.495,A -85,B 0,C 180,E1 11833.613,E2 11833.613} C_VEL
LIN {X 0,Y 564.098,Z 950.024,A -85,B 0,C 180,E1 11836.071,E2 11836.071} C_VEL
LIN {X 0,Y 571.013,Z 904.715,A -85,B 0,C 180,E1 11838.014,E2 11838.014} C_VEL
LIN {X 0,Y 575.564,Z 862.669,A -85,B 0,C 180,E1 11839.337,E2 11839.337} C_VEL
LIN {X 0,Y 555.863,Z 825.589,A -85,B 0,C 180,E1 11842.953,E2 11842.953} C_VEL
LIN {X 0,Y 535.465,Z 794.104,A -85,B 0,C 180,E1 11846.727,E2 11846.727} C_VEL
LIN {X 0,Y 521.237,Z 774.53,A -85,B 0,C 180,E1 11849.687,E2 11849.687} C_VEL
LIN {X 0,Y 517.143,Z 768.569,A -85,B 0,C 180,E1 11850.629,E2 11850.629} C_VEL
LIN {X 0,Y 513.949,Z 763.988,A -85,B 0,C 180,E1 11851.392,E2 11851.392} C_VEL
LIN {X 0,Y 513.723,Z 762.06,A -85,B 0,C 180,E1 11851.558,E2 11851.558} C_VEL
LIN {X 0,Y 513.906,Z 762.06,A -85,B 0,C 180,E1 11857.519,E2 11857.519} C_VEL
LIN {X 0,Y 514.165,Z 762.06,A -85,B 0,C 180,E1 11862.901,E2 11862.901} C_VEL
LIN {X 0,Y 514.392,Z 762.06,A -85,B 0,C 180,E1 11868.125,E2 11868.125} C_VEL
LIN {X 0,Y 514.63,Z 762.06,A -85,B 0,C 180,E1 11873.246,E2 11873.246} C_VEL
LIN {X 0,Y 514.88,Z 762.06,A -85,B 0,C 180,E1 11878.309,E2 11878.309} C_VEL
LIN {X 0,Y 514.836,Z 762.06,A -85,B 0,C 180,E1 11883.687,E2 11883.687} C_VEL
LIN {X 0,Y 514.577,Z 762.06,A -85,B 0,C 180,E1 11888.432,E2 11888.432} C_VEL
LIN {X 0,Y 514.128,Z 762.06,A -85,B 0,C 180,E1 11894.091,E2 11894.091} C_VEL
LIN {X 0,Y 513.895,Z 762.06,A -85,B 0,C 180,E1 11900.649,E2 11900.649} C_VEL
LIN {X 0,Y 513.871,Z 762.06,A -85,B 0,C 180,E1 11906.159,E2 11906.159} C_VEL
LIN {X 0,Y 513.799,Z 762.574,A -85,B 0,C 180,E1 11908.954,E2 11908.954} C_VEL
LIN {X 0,Y 516.02,Z 767.544,A -85,B 0,C 180,E1 11909.539,E2 11909.539} C_VEL
LIN {X 0,Y 518.944,Z 770.816,A -85,B 0,C 180,E1 11910.197,E2 11910.197} C_VEL
LIN {X 0,Y 537.797,Z 797.641,A -85,B 0,C 180,E1 11914.175,E2 11914.175} C_VEL
LIN {X 0,Y 556.903,Z 829.001,A -85,B 0,C 180,E1 11917.928,E2 11917.928} C_VEL
LIN {X 0,Y 573.683,Z 864.021,A -85,B 0,C 180,E1 11921.471,E2 11921.471} C_VEL
LIN {X 0,Y 566.919,Z 909.931,A -85,B 0,C 180,E1 11923.239,E2 11923.239} C_VEL
LIN {X 0,Y 558.295,Z 957.301,A -85,B 0,C 180,E1 11925.812,E2 11925.812} C_VEL
LIN {X 0,Y 549.455,Z 998.678,A -85,B 0,C 180,E1 11928.824,E2 11928.824} C_VEL
LIN {X 0,Y 540.411,Z 1038.165,A -85,B 0,C 180,E1 11932.546,E2 11932.546} C_VEL
LIN {X 0,Y 532.175,Z 1072.73,A -85,B 0,C 180,E1 11936.736,E2 11936.736} C_VEL
LIN {X 0,Y 525.213,Z 1103.84,A -85,B 0,C 180,E1 11941.512,E2 11941.512} C_VEL
LIN {X 0,Y 520.422,Z 1129.114,A -85,B 0,C 180,E1 11946.47,E2 11946.47} C_VEL
LIN {X 0,Y 517.334,Z 1149.877,A -85,B 0,C 180,E1 11951.756,E2 11951.756} C_VEL
LIN {X 0,Y 515.821,Z 1163.531,A -85,B 0,C 180,E1 11956.447,E2 11956.447} C_VEL
LIN {X 0,Y 515.127,Z 1173.598,A -85,B 0,C 180,E1 11961.567,E2 11961.567} C_VEL
LIN {X 0,Y 514.873,Z 1178.921,A -85,B 0,C 180,E1 11966.636,E2 11966.636} C_VEL
LIN {X 0,Y 514.99,Z 1179.656,A -85,B 0,C 180,E1 11971.682,E2 11971.682} C_VEL
LIN {X 0,Y 515.103,Z 1175.855,A -85,B 0,C 180,E1 11976.74,E2 11976.74} C_VEL
LIN {X 0,Y 515.524,Z 1167.195,A -85,B 0,C 180,E1 11981.841,E2 11981.841} C_VEL
LIN {X 0,Y 516.998,Z 1152.413,A -85,B 0,C 180,E1 11987.372,E2 11987.372} C_VEL
LIN {X 0,Y 519.762,Z 1132.615,A -85,B 0,C 180,E1 11992.658,E2 11992.658} C_VEL
LIN {X 0,Y 524.533,Z 1107.086,A -85,B 0,C 180,E1 11997.817,E2 11997.817} C_VEL
LIN {X 0,Y 531.369,Z 1076.124,A -85,B 0,C 180,E1 12002.707,E2 12002.707} C_VEL
LIN {X 0,Y 539.722,Z 1040.907,A -85,B 0,C 180,E1 12007.074,E2 12007.074} C_VEL
LIN {X 0,Y 548.539,Z 1002.895,A -85,B 0,C 180,E1 12010.726,E2 12010.726} C_VEL
LIN {X 0,Y 557.57,Z 961.249,A -85,B 0,C 180,E1 12013.839,E2 12013.839} C_VEL
LIN {X 0,Y 565.763,Z 916.728,A -85,B 0,C 180,E1 12016.348,E2 12016.348} C_VEL
LIN {X 0,Y 573.132,Z 867.871,A -85,B 0,C 180,E1 12018.329,E2 12018.329} C_VEL
LIN {X 0,Y 572.886,Z 862.063,A -85,B 0,C 180,E1 12018.616,E2 12018.616} C_VEL
LIN {X 0,Y 556.165,Z 827.562,A -85,B 0,C 180,E1 12022.122,E2 12022.122} C_VEL
LIN {X 0,Y 536.074,Z 794.807,A -85,B 0,C 180,E1 12026.077,E2 12026.077} C_VEL
LIN {X 0,Y 520.999,Z 774.3,A -85,B 0,C 180,E1 12029.211,E2 12029.211} C_VEL
LIN {X 0,Y 517.2,Z 768.647,A -85,B 0,C 180,E1 12030.088,E2 12030.088} C_VEL
LIN {X 0,Y 513.908,Z 763.98,A -85,B 0,C 180,E1 12030.871,E2 12030.871} C_VEL
LIN {X 0,Y 513.666,Z 762.06,A -85,B 0,C 180,E1 12031.097,E2 12031.097} C_VEL
LIN {X 0,Y 513.789,Z 762.06,A -85,B 0,C 180,E1 12035.749,E2 12035.749} C_VEL
LIN {X 0,Y 513.872,Z 762.06,A -85,B 0,C 180,E1 12041.14,E2 12041.14} C_VEL
LIN {X 0,Y 514.206,Z 762.06,A -85,B 0,C 180,E1 12046.414,E2 12046.414} C_VEL
LIN {X 0,Y 514.592,Z 762.06,A -85,B 0,C 180,E1 12051.568,E2 12051.568} C_VEL
LIN {X 0,Y 514.867,Z 762.06,A -85,B 0,C 180,E1 12056.645,E2 12056.645} C_VEL
LIN {X 0,Y 514.894,Z 762.06,A -85,B 0,C 180,E1 12061.691,E2 12061.691} C_VEL
LIN {X 0,Y 514.642,Z 762.06,A -85,B 0,C 180,E1 12066.754,E2 12066.754} C_VEL
LIN {X 0,Y 514.404,Z 762.06,A -85,B 0,C 180,E1 12071.875,E2 12071.875} C_VEL
LIN {X 0,Y 514.25,Z 762.06,A -85,B 0,C 180,E1 12077.096,E2 12077.096} C_VEL
LIN {X 0,Y 514.071,Z 762.06,A -85,B 0,C 180,E1 12082.474,E2 12082.474} C_VEL
LIN {X 0,Y 513.88,Z 762.06,A -85,B 0,C 180,E1 12088.551,E2 12088.551} C_VEL
LIN {X 0,Y 515.742,Z 767.19,A -85,B 0,C 180,E1 12089.079,E2 12089.079} C_VEL
LIN {X 0,Y 518.977,Z 770.784,A -85,B 0,C 180,E1 12089.806,E2 12089.806} C_VEL
LIN {X 0,Y 537.7,Z 797.344,A -85,B 0,C 180,E1 12093.72,E2 12093.72} C_VEL
LIN {X 0,Y 558.399,Z 829.744,A -85,B 0,C 180,E1 12097.495,E2 12097.495} C_VEL
LIN {X 0,Y 576.07,Z 864.007,A -85,B 0,C 180,E1 12100.771,E2 12100.771} C_VEL
LIN {X 0,Y 570.482,Z 908.619,A -85,B 0,C 180,E1 12102.125,E2 12102.125} C_VEL
LIN {X 0,Y 563.743,Z 951.849,A -85,B 0,C 180,E1 12104.023,E2 12104.023} C_VEL
LIN {X 0,Y 555.176,Z 996.35,A -85,B 0,C 180,E1 12106.64,E2 12106.64} C_VEL
LIN {X 0,Y 546.147,Z 1038.643,A -85,B 0,C 180,E1 12109.897,E2 12109.897} C_VEL
LIN {X 0,Y 537.111,Z 1079.228,A -85,B 0,C 180,E1 12113.974,E2 12113.974} C_VEL
LIN {X 0,Y 529.497,Z 1113.547,A -85,B 0,C 180,E1 12118.371,E2 12118.371} C_VEL
LIN {X 0,Y 523.524,Z 1142.546,A -85,B 0,C 180,E1 12123.139,E2 12123.139} C_VEL
LIN {X 0,Y 523.303,Z 1143.56,A -85,B 0,C 180,E1 12123.323,E2 12123.323} C_VEL
LIN {X 0,Y 517.818,Z 1152.443,A -85,B 0,C 180,E1 12124.876,E2 12124.876} C_VEL
LIN {X 0,Y 512.615,Z 1160.659,A -85,B 0,C 180,E1 12126.5,E2 12126.5} C_VEL
LIN {X 0,Y 509.538,Z 1180.287,A -85,B 0,C 180,E1 12131.633,E2 12131.633} C_VEL
LIN {X 0,Y 507.777,Z 1195.371,A -85,B 0,C 180,E1 12137.102,E2 12137.102} C_VEL
LIN {X 0,Y 507.217,Z 1204.735,A -85,B 0,C 180,E1 12142.295,E2 12142.295} C_VEL
LIN {X 0,Y 507.074,Z 1208.89,A -85,B 0,C 180,E1 12146.582,E2 12146.582} C_VEL
LIN {X 0,Y 507.254,Z 1209.666,A -85,B 0,C 180,E1 12151.706,E2 12151.706} C_VEL
LIN {X 0,Y 507.195,Z 1205.911,A -85,B 0,C 180,E1 12156.844,E2 12156.844} C_VEL
LIN {X 0,Y 507.614,Z 1197.297,A -85,B 0,C 180,E1 12162.027,E2 12162.027} C_VEL
LIN {X 0,Y 509.005,Z 1183.703,A -85,B 0,C 180,E1 12167.269,E2 12167.269} C_VEL
LIN {X 0,Y 511.874,Z 1164.743,A -85,B 0,C 180,E1 12172.567,E2 12172.567} C_VEL
LIN {X 0,Y 516.799,Z 1139.219,A -85,B 0,C 180,E1 12177.893,E2 12177.893} C_VEL
LIN {X 0,Y 523.483,Z 1108.743,A -85,B 0,C 180,E1 12182.768,E2 12182.768} C_VEL
LIN {X 0,Y 531.899,Z 1072.397,A -85,B 0,C 180,E1 12187.294,E2 12187.294} C_VEL
LIN {X 0,Y 540.961,Z 1033.47,A -85,B 0,C 180,E1 12191.092,E2 12191.092} C_VEL
LIN {X 0,Y 550.811,Z 988.676,A -85,B 0,C 180,E1 12194.445,E2 12194.445} C_VEL
LIN {X 0,Y 559.156,Z 945.873,A -85,B 0,C 180,E1 12196.858,E2 12196.858} C_VEL
LIN {X 0,Y 566.085,Z 901.811,A -85,B 0,C 180,E1 12198.708,E2 12198.708} C_VEL
LIN {X 0,Y 570.019,Z 866.172,A -85,B 0,C 180,E1 12199.85,E2 12199.85} C_VEL
LIN {X 0,Y 550.672,Z 829.04,A -85,B 0,C 180,E1 12203.58,E2 12203.58} C_VEL
LIN {X 0,Y 529.136,Z 795.659,A -85,B 0,C 180,E1 12207.739,E2 12207.739} C_VEL
LIN {X 0,Y 513.906,Z 775.011,A -85,B 0,C 180,E1 12211.089,E2 12211.089} C_VEL
LIN {X 0,Y 509.541,Z 768.75,A -85,B 0,C 180,E1 12212.166,E2 12212.166} C_VEL
LIN {X 0,Y 506.127,Z 764.097,A -85,B 0,C 180,E1 12213.042,E2 12213.042} C_VEL
LIN {X 0,Y 505.875,Z 762.06,A -85,B 0,C 180,E1 12213.258,E2 12213.258} C_VEL
LIN {X 0,Y 506.049,Z 762.06,A -85,B 0,C 180,E1 12218.994,E2 12218.994} C_VEL
LIN {X 0,Y 506.301,Z 762.06,A -85,B 0,C 180,E1 12224.41,E2 12224.41} C_VEL
LIN {X 0,Y 506.581,Z 762.06,A -85,B 0,C 180,E1 12229.854,E2 12229.854} C_VEL
LIN {X 0,Y 506.833,Z 762.06,A -85,B 0,C 180,E1 12234.859,E2 12234.859} C_VEL
LIN {X 0,Y 507.133,Z 762.06,A -85,B 0,C 180,E1 12239.99,E2 12239.99} C_VEL
LIN {X 0,Y 506.872,Z 762.06,A -85,B 0,C 180,E1 12245.121,E2 12245.121} C_VEL
LIN {X 0,Y 506.55,Z 762.06,A -85,B 0,C 180,E1 12250.299,E2 12250.299} C_VEL
LIN {X 0,Y 506.108,Z 762.06,A -85,B 0,C 180,E1 12255.576,E2 12255.576} C_VEL
LIN {X 0,Y 505.952,Z 762.06,A -85,B 0,C 180,E1 12260.989,E2 12260.989} C_VEL
LIN {X 0,Y 505.885,Z 762.06,A -85,B 0,C 180,E1 12267.249,E2 12267.249} C_VEL
LIN {X 0,Y 507.693,Z 767.08,A -85,B 0,C 180,E1 12267.806,E2 12267.806} C_VEL
LIN {X 0,Y 511.12,Z 770.706,A -85,B 0,C 180,E1 12268.638,E2 12268.638} C_VEL
LIN {X 0,Y 529.827,Z 796.966,A -85,B 0,C 180,E1 12272.852,E2 12272.852} C_VEL
LIN {X 0,Y 548.354,Z 826.901,A -85,B 0,C 180,E1 12276.681,E2 12276.681} C_VEL
LIN {X 0,Y 565.374,Z 861.28,A -85,B 0,C 180,E1 12280.366,E2 12280.366} C_VEL
LIN {X 0,Y 567.959,Z 868.817,A -85,B 0,C 180,E1 12281.024,E2 12281.024} C_VEL
LIN {X 0,Y 560.55,Z 915.528,A -85,B 0,C 180,E1 12282.901,E2 12282.901} C_VEL
LIN {X 0,Y 551.801,Z 961.039,A -85,B 0,C 180,E1 12285.448,E2 12285.448} C_VEL
LIN {X 0,Y 542.067,Z 1004.366,A -85,B 0,C 180,E1 12288.718,E2 12288.718} C_VEL
LIN {X 0,Y 533.158,Z 1041.352,A -85,B 0,C 180,E1 12292.324,E2 12292.324} C_VEL
LIN {X 0,Y 524.336,Z 1076.986,A -85,B 0,C 180,E1 12296.8,E2 12296.8} C_VEL
LIN {X 0,Y 517.392,Z 1106.622,A -85,B 0,C 180,E1 12301.568,E2 12301.568} C_VEL
LIN {X 0,Y 512.134,Z 1133.249,A -85,B 0,C 180,E1 12307.046,E2 12307.046} C_VEL
LIN {X 0,Y 509.29,Z 1152.078,A -85,B 0,C 180,E1 12312.153,E2 12312.153} C_VEL
LIN {X 0,Y 507.776,Z 1165.474,A -85,B 0,C 180,E1 12317.104,E2 12317.104} C_VEL
LIN {X 0,Y 507.238,Z 1174.802,A -85,B 0,C 180,E1 12322.297,E2 12322.297} C_VEL
LIN {X 0,Y 506.984,Z 1178.918,A -85,B 0,C 180,E1 12326.583,E2 12326.583} C_VEL
LIN {X 0,Y 507.095,Z 1179.656,A -85,B 0,C 180,E1 12331.708,E2 12331.708} C_VEL
LIN {X 0,Y 507.204,Z 1175.856,A -85,B 0,C 180,E1 12336.845,E2 12336.845} C_VEL
LIN {X 0,Y 507.668,Z 1167.194,A -85,B 0,C 180,E1 12342.027,E2 12342.027} C_VEL
LIN {X 0,Y 509.077,Z 1153.56,A -85,B 0,C 180,E1 12347.268,E2 12347.268} C_VEL
LIN {X 0,Y 511.892,Z 1134.559,A -85,B 0,C 180,E1 12352.568,E2 12352.568} C_VEL
LIN {X 0,Y 516.83,Z 1109.013,A -85,B 0,C 180,E1 12357.893,E2 12357.893} C_VEL
LIN {X 0,Y 523.726,Z 1079.539,A -85,B 0,C 180,E1 12362.752,E2 12362.752} C_VEL
LIN {X 0,Y 532.46,Z 1044.008,A -85,B 0,C 180,E1 12367.283,E2 12367.283} C_VEL
LIN {X 0,Y 541.23,Z 1008.412,A -85,B 0,C 180,E1 12370.838,E2 12370.838} C_VEL
LIN {X 0,Y 550.551,Z 967.107,A -85,B 0,C 180,E1 12374.039,E2 12374.039} C_VEL
LIN {X 0,Y 559.387,Z 922.211,A -85,B 0,C 180,E1 12376.689,E2 12376.689} C_VEL
LIN {X 0,Y 567.098,Z 873.659,A -85,B 0,C 180,E1 12378.731,E2 12378.731} C_VEL
LIN {X 0,Y 567.547,Z 866.15,A -85,B 0,C 180,E1 12379.06,E2 12379.06} C_VEL
LIN {X 0,Y 551.375,Z 832.267,A -85,B 0,C 180,E1 12382.599,E2 12382.599} C_VEL
LIN {X 0,Y 532.659,Z 801.109,A -85,B 0,C 180,E1 12386.452,E2 12386.452} C_VEL
LIN {X 0,Y 514.084,Z 775.181,A -85,B 0,C 180,E1 12390.52,E2 12390.52} C_VEL
LIN {X 0,Y 509.097,Z 768.454,A -85,B 0,C 180,E1 12391.737,E2 12391.737} C_VEL
LIN {X 0,Y 506.007,Z 763.986,A -85,B 0,C 180,E1 12392.537,E2 12392.537} C_VEL
LIN {X 0,Y 505.768,Z 762.06,A -85,B 0,C 180,E1 12392.697,E2 12392.697} C_VEL
LIN {X 0,Y 505.893,Z 762.06,A -85,B 0,C 180,E1 12399.009,E2 12399.009} C_VEL
LIN {X 0,Y 506.118,Z 762.06,A -85,B 0,C 180,E1 12404.425,E2 12404.425} C_VEL
LIN {X 0,Y 506.602,Z 762.06,A -85,B 0,C 180,E1 12409.85,E2 12409.85} C_VEL
LIN {X 0,Y 506.812,Z 762.06,A -85,B 0,C 180,E1 12414.879,E2 12414.879} C_VEL
LIN {X 0,Y 507.153,Z 762.06,A -85,B 0,C 180,E1 12420.01,E2 12420.01} C_VEL
LIN {X 0,Y 506.822,Z 762.06,A -85,B 0,C 180,E1 12425.141,E2 12425.141} C_VEL
LIN {X 0,Y 506.588,Z 762.06,A -85,B 0,C 180,E1 12430.319,E2 12430.319} C_VEL
LIN {X 0,Y 506.367,Z 762.06,A -85,B 0,C 180,E1 12435.588,E2 12435.588} C_VEL
LIN {X 0,Y 506.202,Z 762.06,A -85,B 0,C 180,E1 12440.999,E2 12440.999} C_VEL
LIN {X 0,Y 506.007,Z 762.561,A -85,B 0,C 180,E1 12446.913,E2 12446.913} C_VEL
LIN {X 0,Y 508.249,Z 767.573,A -85,B 0,C 180,E1 12447.55,E2 12447.55} C_VEL
LIN {X 0,Y 511.295,Z 770.951,A -85,B 0,C 180,E1 12448.288,E2 12448.288} C_VEL
LIN {X 0,Y 529.735,Z 796.625,A -85,B 0,C 180,E1 12452.401,E2 12452.401} C_VEL
LIN {X 0,Y 551.108,Z 829.845,A -85,B 0,C 180,E1 12456.509,E2 12456.509} C_VEL
LIN {X 0,Y 569.052,Z 864.282,A -85,B 0,C 180,E1 12459.968,E2 12459.968} C_VEL
LIN {X 0,Y 570.408,Z 868.456,A -85,B 0,C 180,E1 12460.282,E2 12460.282} C_VEL
LIN {X 0,Y 564.438,Z 912.988,A -85,B 0,C 180,E1 12461.691,E2 12461.691} C_VEL
LIN {X 0,Y 556.807,Z 958.457,A -85,B 0,C 180,E1 12463.787,E2 12463.787} C_VEL
LIN {X 0,Y 548.146,Z 1001.629,A -85,B 0,C 180,E1 12466.433,E2 12466.433} C_VEL
LIN {X 0,Y 538.616,Z 1043.599,A -85,B 0,C 180,E1 12469.813,E2 12469.813} C_VEL
LIN {X 0,Y 529.548,Z 1082.708,A -85,B 0,C 180,E1 12473.869,E2 12473.869} C_VEL
LIN {X 0,Y 521.424,Z 1117.716,A -85,B 0,C 180,E1 12478.556,E2 12478.556} C_VEL
LIN {X 0,Y 515.621,Z 1145.14,A -85,B 0,C 180,E1 12483.203,E2 12483.203} C_VEL
LIN {X 0,Y 512.615,Z 1160.659,A -85,B 0,C 180,E1 12486.5,E2 12486.5} C_VEL
LIN {X 0,Y 507.476,Z 1168.371,A -85,B 0,C 180,E1 12488.173,E2 12488.173} C_VEL
LIN {X 0,Y 502.468,Z 1175.411,A -85,B 0,C 180,E1 12489.911,E2 12489.911} C_VEL
LIN {X 0,Y 500.33,Z 1192.216,A -85,B 0,C 180,E1 12495.546,E2 12495.546} C_VEL
LIN {X 0,Y 499.434,Z 1202.212,A -85,B 0,C 180,E1 12500.42,E2 12500.42} C_VEL
LIN {X 0,Y 499.152,Z 1207.642,A -85,B 0,C 180,E1 12504.788,E2 12504.788} C_VEL
LIN {X 0,Y 499.262,Z 1210,A -85,B 0,C 180,E1 12509.999,E2 12509.999} C_VEL
LIN {X 0,Y 499.18,Z 1207.644,A -85,B 0,C 180,E1 12515.21,E2 12515.21} C_VEL
LIN {X 0,Y 499.525,Z 1200.655,A -85,B 0,C 180,E1 12520.457,E2 12520.457} C_VEL
LIN {X 0,Y 500.633,Z 1188.849,A -85,B 0,C 180,E1 12525.762,E2 12525.762} C_VEL
LIN {X 0,Y 503.091,Z 1171.689,A -85,B 0,C 180,E1 12531.126,E2 12531.126} C_VEL
LIN {X 0,Y 507.422,Z 1148.395,A -85,B 0,C 180,E1 12536.531,E2 12536.531} C_VEL
LIN {X 0,Y 513.62,Z 1120.71,A -85,B 0,C 180,E1 12541.431,E2 12541.431} C_VEL
LIN {X 0,Y 522.241,Z 1084.744,A -85,B 0,C 180,E1 12546.383,E2 12546.383} C_VEL
LIN {X 0,Y 531.461,Z 1046.959,A -85,B 0,C 180,E1 12550.424,E2 12550.424} C_VEL
LIN {X 0,Y 541.353,Z 1005.29,A -85,B 0,C 180,E1 12553.881,E2 12553.881} C_VEL
LIN {X 0,Y 550.294,Z 962.809,A -85,B 0,C 180,E1 12556.58,E2 12556.58} C_VEL
LIN {X 0,Y 558.658,Z 915.208,A -85,B 0,C 180,E1 12558.832,E2 12558.832} C_VEL
LIN {X 0,Y 564.441,Z 869.543,A -85,B 0,C 180,E1 12560.388,E2 12560.388} C_VEL
LIN {X 0,Y 546.286,Z 834.183,A -85,B 0,C 180,E1 12564.045,E2 12564.045} C_VEL
LIN {X 0,Y 525.728,Z 801.77,A -85,B 0,C 180,E1 12568.173,E2 12568.173} C_VEL
LIN {X 0,Y 506.869,Z 775.698,A -85,B 0,C 180,E1 12572.53,E2 12572.53} C_VEL
LIN {X 0,Y 501.634,Z 768.701,A -85,B 0,C 180,E1 12573.914,E2 12573.914} C_VEL
LIN {X 0,Y 498.242,Z 764.068,A -85,B 0,C 180,E1 12574.867,E2 12574.867} C_VEL
LIN {X 0,Y 498.004,Z 762.06,A -85,B 0,C 180,E1 12575.048,E2 12575.048} C_VEL
LIN {X 0,Y 498.204,Z 762.06,A -85,B 0,C 180,E1 12580.502,E2 12580.502} C_VEL
LIN {X 0,Y 498.448,Z 762.06,A -85,B 0,C 180,E1 12585.955,E2 12585.955} C_VEL
LIN {X 0,Y 498.706,Z 762.06,A -85,B 0,C 180,E1 12591.277,E2 12591.277} C_VEL
LIN {X 0,Y 498.984,Z 762.06,A -85,B 0,C 180,E1 12596.518,E2 12596.518} C_VEL
LIN {X 0,Y 499.06,Z 762.06,A -85,B 0,C 180,E1 12601.725,E2 12601.725} C_VEL
LIN {X 0,Y 498.839,Z 762.06,A -85,B 0,C 180,E1 12606.949,E2 12606.949} C_VEL
LIN {X 0,Y 498.47,Z 762.06,A -85,B 0,C 180,E1 12612.24,E2 12612.24} C_VEL
LIN {X 0,Y 498.087,Z 762.06,A -85,B 0,C 180,E1 12617.648,E2 12617.648} C_VEL
LIN {X 0,Y 498.001,Z 762.06,A -85,B 0,C 180,E1 12623.219,E2 12623.219} C_VEL
LIN {X 0,Y 497.989,Z 762.201,A -85,B 0,C 180,E1 12625.427,E2 12625.427} C_VEL
LIN {X 0,Y 499.837,Z 767.079,A -85,B 0,C 180,E1 12626.031,E2 12626.031} C_VEL
LIN {X 0,Y 503.441,Z 770.9,A -85,B 0,C 180,E1 12626.985,E2 12626.985} C_VEL
LIN {X 0,Y 519.232,Z 792.786,A -85,B 0,C 180,E1 12630.844,E2 12630.844} C_VEL
LIN {X 0,Y 537.015,Z 819.849,A -85,B 0,C 180,E1 12634.747,E2 12634.747} C_VEL
LIN {X 0,Y 554.526,Z 853.014,A -85,B 0,C 180,E1 12638.607,E2 12638.607} C_VEL
LIN {X 0,Y 562.368,Z 870.85,A -85,B 0,C 180,E1 12640.459,E2 12640.459} C_VEL
LIN {X 0,Y 554.728,Z 918.19,A -85,B 0,C 180,E1 12642.414,E2 12642.414} C_VEL
LIN {X 0,Y 546.095,Z 961.296,A -85,B 0,C 180,E1 12644.855,E2 12644.855} C_VEL
LIN {X 0,Y 535.972,Z 1004.624,A -85,B 0,C 180,E1 12648.143,E2 12648.143} C_VEL
LIN {X 0,Y 526.37,Z 1042.857,A -85,B 0,C 180,E1 12651.923,E2 12651.923} C_VEL
LIN {X 0,Y 517.093,Z 1078.821,A -85,B 0,C 180,E1 12656.525,E2 12656.525} C_VEL
LIN {X 0,Y 510.047,Z 1107.27,A -85,B 0,C 180,E1 12661.199,E2 12661.199} C_VEL
LIN {X 0,Y 504.264,Z 1134.917,A -85,B 0,C 180,E1 12667.073,E2 12667.073} C_VEL
LIN {X 0,Y 501.277,Z 1153.835,A -85,B 0,C 180,E1 12672.456,E2 12672.456} C_VEL
LIN {X 0,Y 499.735,Z 1167.391,A -85,B 0,C 180,E1 12677.781,E2 12677.781} C_VEL
LIN {X 0,Y 499.274,Z 1175.96,A -85,B 0,C 180,E1 12683.047,E2 12683.047} C_VEL
LIN {X 0,Y 499.009,Z 1179.675,A -85,B 0,C 180,E1 12688.266,E2 12688.266} C_VEL
LIN {X 0,Y 499.123,Z 1179.243,A -85,B 0,C 180,E1 12692.826,E2 12692.826} C_VEL
LIN {X 0,Y 499.39,Z 1174.67,A -85,B 0,C 180,E1 12697.827,E2 12697.827} C_VEL
LIN {X 0,Y 499.979,Z 1165.27,A -85,B 0,C 180,E1 12703.102,E2 12703.102} C_VEL
LIN {X 0,Y 501.522,Z 1151.812,A -85,B 0,C 180,E1 12708.131,E2 12708.131} C_VEL
LIN {X 0,Y 504.544,Z 1133.002,A -85,B 0,C 180,E1 12713.289,E2 12713.289} C_VEL
LIN {X 0,Y 510.507,Z 1105.439,A -85,B 0,C 180,E1 12719.06,E2 12719.06} C_VEL
LIN {X 0,Y 518.053,Z 1074.972,A -85,B 0,C 180,E1 12723.93,E2 12723.93} C_VEL
LIN {X 0,Y 527.011,Z 1040.572,A -85,B 0,C 180,E1 12728.247,E2 12728.247} C_VEL
LIN {X 0,Y 536.579,Z 1002.474,A -85,B 0,C 180,E1 12731.941,E2 12731.941} C_VEL
LIN {X 0,Y 545.915,Z 962.404,A -85,B 0,C 180,E1 12734.969,E2 12734.969} C_VEL
LIN {X 0,Y 554.769,Z 917.707,A -85,B 0,C 180,E1 12737.522,E2 12737.522} C_VEL
LIN {X 0,Y 562.153,Z 870.168,A -85,B 0,C 180,E1 12739.51,E2 12739.51} C_VEL
LIN {X 0,Y 546.01,Z 835.852,A -85,B 0,C 180,E1 12743.202,E2 12743.202} C_VEL
LIN {X 0,Y 528.32,Z 806.126,A -85,B 0,C 180,E1 12747.03,E2 12747.03} C_VEL
LIN {X 0,Y 511.711,Z 782.341,A -85,B 0,C 180,E1 12750.794,E2 12750.794} C_VEL
LIN {X 0,Y 505.827,Z 774.782,A -85,B 0,C 180,E1 12752.25,E2 12752.25} C_VEL
LIN {X 0,Y 501.798,Z 768.847,A -85,B 0,C 180,E1 12753.334,E2 12753.334} C_VEL
LIN {X 0,Y 498.173,Z 764.099,A -85,B 0,C 180,E1 12754.342,E2 12754.342} C_VEL
LIN {X 0,Y 497.91,Z 762.06,A -85,B 0,C 180,E1 12754.575,E2 12754.575} C_VEL
LIN {X 0,Y 498.025,Z 762.06,A -85,B 0,C 180,E1 12760.516,E2 12760.516} C_VEL
LIN {X 0,Y 498.343,Z 762.06,A -85,B 0,C 180,E1 12766.011,E2 12766.011} C_VEL
LIN {X 0,Y 498.746,Z 762.06,A -85,B 0,C 180,E1 12771.298,E2 12771.298} C_VEL
LIN {X 0,Y 499.043,Z 762.06,A -85,B 0,C 180,E1 12777.796,E2 12777.796} C_VEL
LIN {X 0,Y 499.028,Z 762.06,A -85,B 0,C 180,E1 12782.158,E2 12782.158} C_VEL
LIN {X 0,Y 498.804,Z 762.06,A -85,B 0,C 180,E1 12786.969,E2 12786.969} C_VEL
LIN {X 0,Y 498.556,Z 762.06,A -85,B 0,C 180,E1 12792.258,E2 12792.258} C_VEL
LIN {X 0,Y 498.372,Z 762.06,A -85,B 0,C 180,E1 12797.659,E2 12797.659} C_VEL
LIN {X 0,Y 498.165,Z 762.06,A -85,B 0,C 180,E1 12803.232,E2 12803.232} C_VEL
LIN {X 0,Y 498.146,Z 762.509,A -85,B 0,C 180,E1 12805.092,E2 12805.092} C_VEL
LIN {X 0,Y 500.328,Z 767.522,A -85,B 0,C 180,E1 12805.776,E2 12805.776} C_VEL
LIN {X 0,Y 503.402,Z 770.529,A -85,B 0,C 180,E1 12806.577,E2 12806.577} C_VEL
LIN {X 0,Y 507.815,Z 776.253,A -85,B 0,C 180,E1 12807.715,E2 12807.715} C_VEL
LIN {X 0,Y 528.957,Z 806.597,A -85,B 0,C 180,E1 12812.516,E2 12812.516} C_VEL
LIN {X 0,Y 549.76,Z 840.271,A -85,B 0,C 180,E1 12816.656,E2 12816.656} C_VEL
LIN {X 0,Y 564.998,Z 870.828,A -85,B 0,C 180,E1 12819.731,E2 12819.731} C_VEL
LIN {X 0,Y 558.698,Z 915.289,A -85,B 0,C 180,E1 12821.181,E2 12821.181} C_VEL
LIN {X 0,Y 550.754,Z 960.704,A -85,B 0,C 180,E1 12823.314,E2 12823.314} C_VEL
LIN {X 0,Y 541.79,Z 1003.367,A -85,B 0,C 180,E1 12825.975,E2 12825.975} C_VEL
LIN {X 0,Y 531.884,Z 1045.141,A -85,B 0,C 180,E1 12829.406,E2 12829.406} C_VEL
LIN {X 0,Y 522.701,Z 1082.946,A -85,B 0,C 180,E1 12833.393,E2 12833.393} C_VEL
LIN {X 0,Y 514.067,Z 1118.518,A -85,B 0,C 180,E1 12838.233,E2 12838.233} C_VEL
LIN {X 0,Y 507.71,Z 1147.301,A -85,B 0,C 180,E1 12843.247,E2 12843.247} C_VEL
LIN {X 0,Y 503.277,Z 1170.509,A -85,B 0,C 180,E1 12848.567,E2 12848.567} C_VEL
LIN {X 0,Y 502.468,Z 1175.411,A -85,B 0,C 180,E1 12849.911,E2 12849.911} C_VEL
LIN {X 0,Y 497.708,Z 1181.897,A -85,B 0,C 180,E1 12851.696,E2 12851.696} C_VEL
LIN {X 0,Y 492.999,Z 1187.711,A -85,B 0,C 180,E1 12853.54,E2 12853.54} C_VEL
LIN {X 0,Y 491.801,Z 1199.088,A -85,B 0,C 180,E1 12858.479,E2 12858.479} C_VEL
LIN {X 0,Y 491.402,Z 1205.908,A -85,B 0,C 180,E1 12862.934,E2 12862.934} C_VEL
LIN {X 0,Y 491.218,Z 1209.665,A -85,B 0,C 180,E1 12868.236,E2 12868.236} C_VEL
LIN {X 0,Y 491.454,Z 1209.666,A -85,B 0,C 180,E1 12871.761,E2 12871.761} C_VEL
LIN {X 0,Y 491.409,Z 1205.911,A -85,B 0,C 180,E1 12877.065,E2 12877.065} C_VEL
LIN {X 0,Y 491.898,Z 1197.291,A -85,B 0,C 180,E1 12882.417,E2 12882.417} C_VEL
LIN {X 0,Y 493.499,Z 1183.701,A -85,B 0,C 180,E1 12887.83,E2 12887.83} C_VEL
LIN {X 0,Y 496.759,Z 1164.733,A -85,B 0,C 180,E1 12893.293,E2 12893.293} C_VEL
LIN {X 0,Y 502.117,Z 1138.678,A -85,B 0,C 180,E1 12898.784,E2 12898.784} C_VEL
LIN {X 0,Y 509.5,Z 1108.445,A -85,B 0,C 180,E1 12903.746,E2 12903.746} C_VEL
LIN {X 0,Y 518.904,Z 1071.208,A -85,B 0,C 180,E1 12908.483,E2 12908.483} C_VEL
LIN {X 0,Y 528.676,Z 1032.79,A -85,B 0,C 180,E1 12912.279,E2 12912.279} C_VEL
LIN {X 0,Y 539.386,Z 987.544,A -85,B 0,C 180,E1 12915.704,E2 12915.704} C_VEL
LIN {X 0,Y 548.592,Z 942.839,A -85,B 0,C 180,E1 12918.221,E2 12918.221} C_VEL
LIN {X 0,Y 555.873,Z 899.972,A -85,B 0,C 180,E1 12919.992,E2 12919.992} C_VEL
LIN {X 0,Y 558.947,Z 872.957,A -85,B 0,C 180,E1 12920.924,E2 12920.924} C_VEL
LIN {X 0,Y 541.468,Z 838.53,A -85,B 0,C 180,E1 12924.593,E2 12924.593} C_VEL
LIN {X 0,Y 522.353,Z 807.861,A -85,B 0,C 180,E1 12928.613,E2 12928.613} C_VEL
LIN {X 0,Y 504.363,Z 782.673,A -85,B 0,C 180,E1 12932.865,E2 12932.865} C_VEL
LIN {X 0,Y 498.625,Z 775.311,A -85,B 0,C 180,E1 12934.407,E2 12934.407} C_VEL
LIN {X 0,Y 494.37,Z 769.044,A -85,B 0,C 180,E1 12935.66,E2 12935.66} C_VEL
LIN {X 0,Y 490.432,Z 764.341,A -85,B 0,C 180,E1 12936.857,E2 12936.857} C_VEL
LIN {X 0,Y 490.097,Z 762.06,A -85,B 0,C 180,E1 12937.058,E2 12937.058} C_VEL
LIN {X 0,Y 490.361,Z 762.06,A -85,B 0,C 180,E1 12942.802,E2 12942.802} C_VEL
LIN {X 0,Y 490.738,Z 762.06,A -85,B 0,C 180,E1 12949.344,E2 12949.344} C_VEL
LIN {X 0,Y 491.003,Z 762.06,A -85,B 0,C 180,E1 12954.693,E2 12954.693} C_VEL
LIN {X 0,Y 491.339,Z 762.06,A -85,B 0,C 180,E1 12959.99,E2 12959.99} C_VEL
LIN {X 0,Y 491.061,Z 762.06,A -85,B 0,C 180,E1 12965.286,E2 12965.286} C_VEL
LIN {X 0,Y 490.704,Z 762.06,A -85,B 0,C 180,E1 12970.636,E2 12970.636} C_VEL
LIN {X 0,Y 490.185,Z 762.06,A -85,B 0,C 180,E1 12977.131,E2 12977.131} C_VEL
LIN {X 0,Y 490.104,Z 762.368,A -85,B 0,C 180,E1 12983.399,E2 12983.399} C_VEL
LIN {X 0,Y 492.07,Z 767.3,A -85,B 0,C 180,E1 12984.102,E2 12984.102} C_VEL
LIN {X 0,Y 495.62,Z 770.699,A -85,B 0,C 180,E1 12985.127,E2 12985.127} C_VEL
LIN {X 0,Y 500.102,Z 776.384,A -85,B 0,C 180,E1 12986.392,E2 12986.392} C_VEL
LIN {X 0,Y 519.498,Z 803.97,A -85,B 0,C 180,E1 12991.245,E2 12991.245} C_VEL
LIN {X 0,Y 536.763,Z 832.168,A -85,B 0,C 180,E1 12995.167,E2 12995.167} C_VEL
LIN {X 0,Y 552.905,Z 865.025,A -85,B 0,C 180,E1 12998.972,E2 12998.972} C_VEL
LIN {X 0,Y 556.726,Z 875.376,A -85,B 0,C 180,E1 13000.007,E2 13000.007} C_VEL
LIN {X 0,Y 549.162,Z 919.477,A -85,B 0,C 180,E1 13001.847,E2 13001.847} C_VEL
LIN {X 0,Y 539.964,Z 963.461,A -85,B 0,C 180,E1 13004.378,E2 13004.378} C_VEL
LIN {X 0,Y 529.236,Z 1007.685,A -85,B 0,C 180,E1 13007.797,E2 13007.797} C_VEL
LIN {X 0,Y 519.299,Z 1045.365,A -85,B 0,C 180,E1 13011.626,E2 13011.626} C_VEL
LIN {X 0,Y 510.015,Z 1080.041,A -85,B 0,C 180,E1 13016.153,E2 13016.153} C_VEL
LIN {X 0,Y 502.255,Z 1109.998,A -85,B 0,C 180,E1 13021.225,E2 13021.225} C_VEL
LIN {X 0,Y 496.711,Z 1134.95,A -85,B 0,C 180,E1 13026.704,E2 13026.704} C_VEL
LIN {X 0,Y 493.325,Z 1155.166,A -85,B 0,C 180,E1 13032.624,E2 13032.624} C_VEL
LIN {X 0,Y 491.884,Z 1167.386,A -85,B 0,C 180,E1 13037.583,E2 13037.583} C_VEL
LIN {X 0,Y 491.377,Z 1175.959,A -85,B 0,C 180,E1 13042.935,E2 13042.935} C_VEL
LIN {X 0,Y 491.128,Z 1179.675,A -85,B 0,C 180,E1 13048.238,E2 13048.238} C_VEL
LIN {X 0,Y 491.299,Z 1179.656,A -85,B 0,C 180,E1 13051.763,E2 13051.763} C_VEL
LIN {X 0,Y 491.415,Z 1175.857,A -85,B 0,C 180,E1 13057.066,E2 13057.066} C_VEL
LIN {X 0,Y 491.938,Z 1167.191,A -85,B 0,C 180,E1 13062.418,E2 13062.418} C_VEL
LIN {X 0,Y 493.562,Z 1153.563,A -85,B 0,C 180,E1 13067.829,E2 13067.829} C_VEL
LIN {X 0,Y 496.741,Z 1134.608,A -85,B 0,C 180,E1 13073.296,E2 13073.296} C_VEL
LIN {X 0,Y 502.32,Z 1109.562,A -85,B 0,C 180,E1 13078.773,E2 13078.773} C_VEL
LIN {X 0,Y 509.796,Z 1080.814,A -85,B 0,C 180,E1 13083.648,E2 13083.648} C_VEL
LIN {X 0,Y 519.183,Z 1045.851,A -85,B 0,C 180,E1 13088.225,E2 13088.225} C_VEL
LIN {X 0,Y 529.068,Z 1008.627,A -85,B 0,C 180,E1 13092.023,E2 13092.023} C_VEL
LIN {X 0,Y 539.4,Z 966.084,A -85,B 0,C 180,E1 13095.343,E2 13095.343} C_VEL
LIN {X 0,Y 548.677,Z 921.929,A -85,B 0,C 180,E1 13097.946,E2 13097.946} C_VEL
LIN {X 0,Y 556.641,Z 873.857,A -85,B 0,C 180,E1 13099.993,E2 13099.993} C_VEL
LIN {X 0,Y 541.012,Z 840.07,A -85,B 0,C 180,E1 13103.745,E2 13103.745} C_VEL
LIN {X 0,Y 522.654,Z 808.533,A -85,B 0,C 180,E1 13107.938,E2 13107.938} C_VEL
LIN {X 0,Y 504.119,Z 782.494,A -85,B 0,C 180,E1 13112.39,E2 13112.39} C_VEL
LIN {X 0,Y 498.38,Z 775.09,A -85,B 0,C 180,E1 13113.933,E2 13113.933} C_VEL
LIN {X 0,Y 494.06,Z 768.965,A -85,B 0,C 180,E1 13115.198,E2 13115.198} C_VEL
LIN {X 0,Y 490.281,Z 764.194,A -85,B 0,C 180,E1 13116.356,E2 13116.356} C_VEL
LIN {X 0,Y 489.991,Z 762.06,A -85,B 0,C 180,E1 13116.556,E2 13116.556} C_VEL
LIN {X 0,Y 490.16,Z 762.06,A -85,B 0,C 180,E1 13122.884,E2 13122.884} C_VEL
LIN {X 0,Y 490.719,Z 762.06,A -85,B 0,C 180,E1 13129.364,E2 13129.364} C_VEL
LIN {X 0,Y 490.989,Z 762.06,A -85,B 0,C 180,E1 13134.713,E2 13134.713} C_VEL
LIN {X 0,Y 491.359,Z 762.06,A -85,B 0,C 180,E1 13140.01,E2 13140.01} C_VEL
LIN {X 0,Y 490.998,Z 762.06,A -85,B 0,C 180,E1 13145.307,E2 13145.307} C_VEL
LIN {X 0,Y 490.751,Z 762.06,A -85,B 0,C 180,E1 13150.656,E2 13150.656} C_VEL
LIN {X 0,Y 490.494,Z 762.06,A -85,B 0,C 180,E1 13156.106,E2 13156.106} C_VEL
LIN {X 0,Y 490.245,Z 762.06,A -85,B 0,C 180,E1 13162.373,E2 13162.373} C_VEL
LIN {X 0,Y 490.285,Z 762.632,A -85,B 0,C 180,E1 13163.082,E2 13163.082} C_VEL
LIN {X 0,Y 492.569,Z 767.67,A -85,B 0,C 180,E1 13163.867,E2 13163.867} C_VEL
LIN {X 0,Y 495.736,Z 770.708,A -85,B 0,C 180,E1 13164.774,E2 13164.774} C_VEL
LIN {X 0,Y 500.26,Z 776.42,A -85,B 0,C 180,E1 13166.044,E2 13166.044} C_VEL
LIN {X 0,Y 519.946,Z 804.355,A -85,B 0,C 180,E1 13170.88,E2 13170.88} C_VEL
LIN {X 0,Y 539.162,Z 834.446,A -85,B 0,C 180,E1 13174.931,E2 13174.931} C_VEL
LIN {X 0,Y 556.376,Z 867.499,A -85,B 0,C 180,E1 13178.538,E2 13178.538} C_VEL
LIN {X 0,Y 559.299,Z 875.555,A -85,B 0,C 180,E1 13179.243,E2 13179.243} C_VEL
LIN {X 0,Y 552.546,Z 920.325,A -85,B 0,C 180,E1 13180.773,E2 13180.773} C_VEL
LIN {X 0,Y 544.099,Z 966.087,A -85,B 0,C 180,E1 13182.999,E2 13182.999} C_VEL
LIN {X 0,Y 534.908,Z 1007.378,A -85,B 0,C 180,E1 13185.691,E2 13185.691} C_VEL
LIN {X 0,Y 524.508,Z 1049.396,A -85,B 0,C 180,E1 13189.244,E2 13189.244} C_VEL
LIN {X 0,Y 515.076,Z 1086.245,A -85,B 0,C 180,E1 13193.29,E2 13193.29} C_VEL
LIN {X 0,Y 506.224,Z 1121.466,A -85,B 0,C 180,E1 13198.231,E2 13198.231} C_VEL
LIN {X 0,Y 499.531,Z 1150.33,A -85,B 0,C 180,E1 13203.499,E2 13203.499} C_VEL
LIN {X 0,Y 495.441,Z 1171.683,A -85,B 0,C 180,E1 13208.53,E2 13208.53} C_VEL
LIN {X 0,Y 492.999,Z 1187.711,A -85,B 0,C 180,E1 13213.54,E2 13213.54} C_VEL
LIN {X 0,Y 488.401,Z 1192.819,A -85,B 0,C 180,E1 13215.428,E2 13215.428} C_VEL
LIN {X 0,Y 484.052,Z 1197.255,A -85,B 0,C 180,E1 13217.363,E2 13217.363} C_VEL
LIN {X 0,Y 483.5,Z 1205.908,A -85,B 0,C 180,E1 13222.818,E2 13222.818} C_VEL
LIN {X 0,Y 483.347,Z 1209.665,A -85,B 0,C 180,E1 13228.208,E2 13228.208} C_VEL
LIN {X 0,Y 483.556,Z 1209.666,A -85,B 0,C 180,E1 13231.79,E2 13231.79} C_VEL
LIN {X 0,Y 483.507,Z 1205.911,A -85,B 0,C 180,E1 13237.181,E2 13237.181} C_VEL
LIN {X 0,Y 484.036,Z 1197.287,A -85,B 0,C 180,E1 13242.622,E2 13242.622} C_VEL
LIN {X 0,Y 485.761,Z 1183.7,A -85,B 0,C 180,E1 13248.123,E2 13248.123} C_VEL
LIN {X 0,Y 489.21,Z 1164.463,A -85,B 0,C 180,E1 13253.674,E2 13253.674} C_VEL
LIN {X 0,Y 494.862,Z 1138.406,A -85,B 0,C 180,E1 13259.246,E2 13259.246} C_VEL
LIN {X 0,Y 502.588,Z 1108.171,A -85,B 0,C 180,E1 13264.274,E2 13264.274} C_VEL
LIN {X 0,Y 512.492,Z 1070.847,A -85,B 0,C 180,E1 13269.068,E2 13269.068} C_VEL
LIN {X 0,Y 522.623,Z 1032.271,A -85,B 0,C 180,E1 13272.913,E2 13272.913} C_VEL
LIN {X 0,Y 533.661,Z 987.419,A -85,B 0,C 180,E1 13276.324,E2 13276.324} C_VEL
LIN {X 0,Y 543.241,Z 942.579,A -85,B 0,C 180,E1 13278.856,E2 13278.856} C_VEL
LIN {X 0,Y 550.96,Z 898.359,A -85,B 0,C 180,E1 13280.68,E2 13280.68} C_VEL
LIN {X 0,Y 553.562,Z 876.92,A -85,B 0,C 180,E1 13281.415,E2 13281.415} C_VEL
LIN {X 0,Y 536.639,Z 842.669,A -85,B 0,C 180,E1 13285.168,E2 13285.168} C_VEL
LIN {X 0,Y 518.634,Z 813.5,A -85,B 0,C 180,E1 13289.12,E2 13289.12} C_VEL
LIN {X 0,Y 501.684,Z 789.434,A -85,B 0,C 180,E1 13293.253,E2 13293.253} C_VEL
LIN {X 0,Y 491.583,Z 775.973,A -85,B 0,C 180,E1 13296.137,E2 13296.137} C_VEL
LIN {X 0,Y 487.721,Z 770.181,A -85,B 0,C 180,E1 13297.388,E2 13297.388} C_VEL
LIN {X 0,Y 482.697,Z 764.692,A -85,B 0,C 180,E1 13299.071,E2 13299.071} C_VEL
LIN {X 0,Y 482.275,Z 762.06,A -85,B 0,C 180,E1 13299.352,E2 13299.352} C_VEL
LIN {X 0,Y 482.616,Z 762.06,A -85,B 0,C 180,E1 13306.077,E2 13306.077} C_VEL
LIN {X 0,Y 482.893,Z 762.06,A -85,B 0,C 180,E1 13310.989,E2 13310.989} C_VEL
LIN {X 0,Y 483.175,Z 762.06,A -85,B 0,C 180,E1 13316.404,E2 13316.404} C_VEL
LIN {X 0,Y 483.288,Z 762.06,A -85,B 0,C 180,E1 13321.781,E2 13321.781} C_VEL
LIN {X 0,Y 482.998,Z 762.06,A -85,B 0,C 180,E1 13327.178,E2 13327.178} C_VEL
LIN {X 0,Y 482.594,Z 762.06,A -85,B 0,C 180,E1 13332.649,E2 13332.649} C_VEL
LIN {X 0,Y 482.212,Z 762.06,A -85,B 0,C 180,E1 13338.249,E2 13338.249} C_VEL
LIN {X 0,Y 482.195,Z 762.698,A -85,B 0,C 180,E1 13341.11,E2 13341.11} C_VEL
LIN {X 0,Y 484.492,Z 767.645,A -85,B 0,C 180,E1 13342.005,E2 13342.005} C_VEL
LIN {X 0,Y 487.841,Z 770.63,A -85,B 0,C 180,E1 13343.079,E2 13343.079} C_VEL
LIN {X 0,Y 492.07,Z 776.297,A -85,B 0,C 180,E1 13344.418,E2 13344.418} C_VEL
LIN {X 0,Y 507.905,Z 797.913,A -85,B 0,C 180,E1 13348.786,E2 13348.786} C_VEL
LIN {X 0,Y 526.417,Z 826.494,A -85,B 0,C 180,E1 13353.282,E2 13353.282} C_VEL
LIN {X 0,Y 543.694,Z 860.181,A -85,B 0,C 180,E1 13357.489,E2 13357.489} C_VEL
LIN {X 0,Y 551.215,Z 878.496,A -85,B 0,C 180,E1 13359.479,E2 13359.479} C_VEL
LIN {X 0,Y 543.416,Z 922.188,A -85,B 0,C 180,E1 13361.341,E2 13361.341} C_VEL
LIN {X 0,Y 533.567,Z 966.845,A -85,B 0,C 180,E1 13363.973,E2 13363.973} C_VEL
LIN {X 0,Y 522.765,Z 1009.806,A -85,B 0,C 180,E1 13367.361,E2 13367.361} C_VEL
LIN {X 0,Y 512.387,Z 1047.409,A -85,B 0,C 180,E1 13371.267,E2 13371.267} C_VEL
LIN {X 0,Y 502.885,Z 1081.558,A -85,B 0,C 180,E1 13375.815,E2 13375.815} C_VEL
LIN {X 0,Y 494.752,Z 1111.441,A -85,B 0,C 180,E1 13380.997,E2 13380.997} C_VEL
LIN {X 0,Y 489.218,Z 1135.216,A -85,B 0,C 180,E1 13386.326,E2 13386.326} C_VEL
LIN {X 0,Y 485.587,Z 1155.163,A -85,B 0,C 180,E1 13392.338,E2 13392.338} C_VEL
LIN {X 0,Y 484.037,Z 1167.382,A -85,B 0,C 180,E1 13397.378,E2 13397.378} C_VEL
LIN {X 0,Y 483.48,Z 1175.958,A -85,B 0,C 180,E1 13402.819,E2 13402.819} C_VEL
LIN {X 0,Y 483.225,Z 1179.674,A -85,B 0,C 180,E1 13408.209,E2 13408.209} C_VEL
LIN {X 0,Y 483.393,Z 1179.656,A -85,B 0,C 180,E1 13411.792,E2 13411.792} C_VEL
LIN {X 0,Y 483.52,Z 1175.858,A -85,B 0,C 180,E1 13417.182,E2 13417.182} C_VEL
LIN {X 0,Y 484.083,Z 1167.189,A -85,B 0,C 180,E1 13422.623,E2 13422.623} C_VEL
LIN {X 0,Y 485.791,Z 1153.564,A -85,B 0,C 180,E1 13428.124,E2 13428.124} C_VEL
LIN {X 0,Y 489.232,Z 1134.88,A -85,B 0,C 180,E1 13433.675,E2 13433.675} C_VEL
LIN {X 0,Y 495.125,Z 1109.836,A -85,B 0,C 180,E1 13439.231,E2 13439.231} C_VEL
LIN {X 0,Y 503.121,Z 1080.698,A -85,B 0,C 180,E1 13444.22,E2 13444.22} C_VEL
LIN {X 0,Y 513.189,Z 1044.725,A -85,B 0,C 180,E1 13448.955,E2 13448.955} C_VEL
LIN {X 0,Y 523.251,Z 1008.114,A -85,B 0,C 180,E1 13452.688,E2 13452.688} C_VEL
LIN {X 0,Y 533.572,Z 967.189,A -85,B 0,C 180,E1 13455.9,E2 13455.9} C_VEL
LIN {X 0,Y 543.132,Z 923.342,A -85,B 0,C 180,E1 13458.518,E2 13458.518} C_VEL
LIN {X 0,Y 551.081,Z 877.466,A -85,B 0,C 180,E1 13460.501,E2 13460.501} C_VEL
LIN {X 0,Y 536.004,Z 844.284,A -85,B 0,C 180,E1 13464.307,E2 13464.307} C_VEL
LIN {X 0,Y 519.318,Z 814.905,A -85,B 0,C 180,E1 13468.311,E2 13468.311} C_VEL
LIN {X 0,Y 501.446,Z 789.224,A -85,B 0,C 180,E1 13472.778,E2 13472.778} C_VEL
LIN {X 0,Y 495.079,Z 781.035,A -85,B 0,C 180,E1 13474.536,E2 13474.536} C_VEL
LIN {X 0,Y 491.328,Z 775.811,A -85,B 0,C 180,E1 13475.664,E2 13475.664} C_VEL
LIN {X 0,Y 487.576,Z 770.091,A -85,B 0,C 180,E1 13476.882,E2 13476.882} C_VEL
LIN {X 0,Y 482.582,Z 764.738,A -85,B 0,C 180,E1 13478.547,E2 13478.547} C_VEL
LIN {X 0,Y 482.114,Z 762.06,A -85,B 0,C 180,E1 13478.886,E2 13478.886} C_VEL
LIN {X 0,Y 482.449,Z 762.06,A -85,B 0,C 180,E1 13485.501,E2 13485.501} C_VEL
LIN {X 0,Y 482.918,Z 762.06,A -85,B 0,C 180,E1 13491.01,E2 13491.01} C_VEL
LIN {X 0,Y 483.272,Z 762.06,A -85,B 0,C 180,E1 13496.425,E2 13496.425} C_VEL
LIN {X 0,Y 483.338,Z 762.06,A -85,B 0,C 180,E1 13501.802,E2 13501.802} C_VEL
LIN {X 0,Y 482.971,Z 762.06,A -85,B 0,C 180,E1 13507.199,E2 13507.199} C_VEL
LIN {X 0,Y 482.707,Z 762.06,A -85,B 0,C 180,E1 13512.667,E2 13512.667} C_VEL
LIN {X 0,Y 482.499,Z 762.06,A -85,B 0,C 180,E1 13518.26,E2 13518.26} C_VEL
LIN {X 0,Y 482.442,Z 762.687,A -85,B 0,C 180,E1 13520.821,E2 13520.821} C_VEL
LIN {X 0,Y 484.656,Z 767.54,A -85,B 0,C 180,E1 13521.679,E2 13521.679} C_VEL
LIN {X 0,Y 488.023,Z 770.657,A -85,B 0,C 180,E1 13522.756,E2 13522.756} C_VEL
LIN {X 0,Y 492.201,Z 776.271,A -85,B 0,C 180,E1 13524.071,E2 13524.071} C_VEL
LIN {X 0,Y 508.141,Z 798.05,A -85,B 0,C 180,E1 13528.419,E2 13528.419} C_VEL
LIN {X 0,Y 527.552,Z 827.108,A -85,B 0,C 180,E1 13532.859,E2 13532.859} C_VEL
LIN {X 0,Y 546.578,Z 861.722,A -85,B 0,C 180,E1 13537.014,E2 13537.014} C_VEL
LIN {X 0,Y 553.87,Z 877.637,A -85,B 0,C 180,E1 13538.662,E2 13538.662} C_VEL
LIN {X 0,Y 546.278,Z 925.766,A -85,B 0,C 180,E1 13540.364,E2 13540.364} C_VEL
LIN {X 0,Y 537.557,Z 970.336,A -85,B 0,C 180,E1 13542.628,E2 13542.628} C_VEL
LIN {X 0,Y 527.598,Z 1012.875,A -85,B 0,C 180,E1 13545.506,E2 13545.506} C_VEL
LIN {X 0,Y 517.258,Z 1053.062,A -85,B 0,C 180,E1 13549.035,E2 13549.035} C_VEL
LIN {X 0,Y 506.736,Z 1092.351,A -85,B 0,C 180,E1 13553.543,E2 13553.543} C_VEL
LIN {X 0,Y 498.41,Z 1123.983,A -85,B 0,C 180,E1 13558.195,E2 13558.195} C_VEL
LIN {X 0,Y 491.486,Z 1152.943,A -85,B 0,C 180,E1 13563.674,E2 13563.674} C_VEL
LIN {X 0,Y 487.408,Z 1173.837,A -85,B 0,C 180,E1 13568.795,E2 13568.795} C_VEL
LIN {X 0,Y 485.062,Z 1188.837,A -85,B 0,C 180,E1 13573.716,E2 13573.716} C_VEL
LIN {X 0,Y 484.052,Z 1197.255,A -85,B 0,C 180,E1 13577.363,E2 13577.363} C_VEL
LIN {X 0,Y 482.642,Z 1199.281,A -85,B 0,C 180,E1 13578.359,E2 13578.359} C_VEL
LIN {X 0,Y 475.756,Z 1203.828,A -85,B 0,C 180,E1 13581.094,E2 13581.094} C_VEL
LIN {X 0,Y 475.654,Z 1204.167,A -85,B 0,C 180,E1 13581.356,E2 13581.356} C_VEL
LIN {X 0,Y 475.456,Z 1208.878,A -85,B 0,C 180,E1 13586.355,E2 13586.355} C_VEL
LIN {X 0,Y 475.647,Z 1209.666,A -85,B 0,C 180,E1 13591.82,E2 13591.82} C_VEL
LIN {X 0,Y 475.608,Z 1205.911,A -85,B 0,C 180,E1 13597.3,E2 13597.3} C_VEL
LIN {X 0,Y 476.179,Z 1197.285,A -85,B 0,C 180,E1 13602.834,E2 13602.834} C_VEL
LIN {X 0,Y 478.094,Z 1183.359,A -85,B 0,C 180,E1 13608.509,E2 13608.509} C_VEL
LIN {X 0,Y 481.698,Z 1164.193,A -85,B 0,C 180,E1 13614.067,E2 13614.067} C_VEL
LIN {X 0,Y 487.809,Z 1137.529,A -85,B 0,C 180,E1 13619.837,E2 13619.837} C_VEL
LIN {X 0,Y 495.761,Z 1107.751,A -85,B 0,C 180,E1 13624.838,E2 13624.838} C_VEL
LIN {X 0,Y 506.068,Z 1070.576,A -85,B 0,C 180,E1 13629.661,E2 13629.661} C_VEL
LIN {X 0,Y 516.366,Z 1033.023,A -85,B 0,C 180,E1 13633.447,E2 13633.447} C_VEL
LIN {X 0,Y 527.737,Z 988.365,A -85,B 0,C 180,E1 13636.885,E2 13636.885} C_VEL
LIN {X 0,Y 537.46,Z 944.829,A -85,B 0,C 180,E1 13639.386,E2 13639.386} C_VEL
LIN {X 0,Y 545.619,Z 900,A -85,B 0,C 180,E1 13641.262,E2 13641.262} C_VEL
LIN {X 0,Y 548.002,Z 880.17,A -85,B 0,C 180,E1 13641.979,E2 13641.979} C_VEL
LIN {X 0,Y 531.742,Z 846.797,A -85,B 0,C 180,E1 13645.773,E2 13645.773} C_VEL
LIN {X 0,Y 514.662,Z 818.691,A -85,B 0,C 180,E1 13649.694,E2 13649.694} C_VEL
LIN {X 0,Y 498.845,Z 795.942,A -85,B 0,C 180,E1 13653.695,E2 13653.695} C_VEL
LIN {X 0,Y 488.919,Z 782.683,A -85,B 0,C 180,E1 13656.603,E2 13656.603} C_VEL
LIN {X 0,Y 484.155,Z 776.242,A -85,B 0,C 180,E1 13658.177,E2 13658.177} C_VEL
LIN {X 0,Y 480.168,Z 770.597,A -85,B 0,C 180,E1 13659.618,E2 13659.618} C_VEL
LIN {X 0,Y 474.966,Z 764.759,A -85,B 0,C 180,E1 13661.628,E2 13661.628} C_VEL
LIN {X 0,Y 474.52,Z 762.06,A -85,B 0,C 180,E1 13661.986,E2 13661.986} C_VEL
LIN {X 0,Y 474.764,Z 762.06,A -85,B 0,C 180,E1 13667.117,E2 13667.117} C_VEL
LIN {X 0,Y 475.039,Z 762.06,A -85,B 0,C 180,E1 13672.68,E2 13672.68} C_VEL
LIN {X 0,Y 475.43,Z 762.06,A -85,B 0,C 180,E1 13678.168,E2 13678.168} C_VEL
LIN {X 0,Y 475.38,Z 762.06,A -85,B 0,C 180,E1 13683.634,E2 13683.634} C_VEL
LIN {X 0,Y 474.944,Z 762.06,A -85,B 0,C 180,E1 13689.496,E2 13689.496} C_VEL
LIN {X 0,Y 474.49,Z 762.06,A -85,B 0,C 180,E1 13694.747,E2 13694.747} C_VEL
LIN {X 0,Y 474.339,Z 762.706,A -85,B 0,C 180,E1 13698.465,E2 13698.465} C_VEL
LIN {X 0,Y 476.456,Z 767.49,A -85,B 0,C 180,E1 13699.437,E2 13699.437} C_VEL
LIN {X 0,Y 480.112,Z 770.652,A -85,B 0,C 180,E1 13700.784,E2 13700.784} C_VEL
LIN {X 0,Y 484.271,Z 776.337,A -85,B 0,C 180,E1 13702.278,E2 13702.278} C_VEL
LIN {X 0,Y 496.642,Z 792.751,A -85,B 0,C 180,E1 13706.104,E2 13706.104} C_VEL
LIN {X 0,Y 513.03,Z 816.579,A -85,B 0,C 180,E1 13710.476,E2 13710.476} C_VEL
LIN {X 0,Y 529.095,Z 844.732,A -85,B 0,C 180,E1 13714.537,E2 13714.537} C_VEL
LIN {X 0,Y 543.871,Z 876.987,A -85,B 0,C 180,E1 13718.422,E2 13718.422} C_VEL
LIN {X 0,Y 545.487,Z 883.202,A -85,B 0,C 180,E1 13718.996,E2 13718.996} C_VEL
LIN {X 0,Y 537.775,Z 924.471,A -85,B 0,C 180,E1 13720.801,E2 13720.801} C_VEL
LIN {X 0,Y 527.49,Z 969.132,A -85,B 0,C 180,E1 13723.483,E2 13723.483} C_VEL
LIN {X 0,Y 516.406,Z 1011.506,A -85,B 0,C 180,E1 13726.881,E2 13726.881} C_VEL
LIN {X 0,Y 505.044,Z 1050.942,A -85,B 0,C 180,E1 13731.074,E2 13731.074} C_VEL
LIN {X 0,Y 495.237,Z 1084.549,A -85,B 0,C 180,E1 13735.713,E2 13735.713} C_VEL
LIN {X 0,Y 486.75,Z 1115.233,A -85,B 0,C 180,E1 13741.237,E2 13741.237} C_VEL
LIN {X 0,Y 480.914,Z 1138.873,A -85,B 0,C 180,E1 13746.874,E2 13746.874} C_VEL
LIN {X 0,Y 477.638,Z 1156.554,A -85,B 0,C 180,E1 13752.51,E2 13752.51} C_VEL
LIN {X 0,Y 476.021,Z 1169.16,A -85,B 0,C 180,E1 13758.093,E2 13758.093} C_VEL
LIN {X 0,Y 475.583,Z 1175.957,A -85,B 0,C 180,E1 13762.699,E2 13762.699} C_VEL
LIN {X 0,Y 475.323,Z 1179.674,A -85,B 0,C 180,E1 13768.179,E2 13768.179} C_VEL
LIN {X 0,Y 475.487,Z 1179.656,A -85,B 0,C 180,E1 13771.822,E2 13771.822} C_VEL
LIN {X 0,Y 475.626,Z 1175.859,A -85,B 0,C 180,E1 13777.302,E2 13777.302} C_VEL
LIN {X 0,Y 476.229,Z 1167.188,A -85,B 0,C 180,E1 13782.834,E2 13782.834} C_VEL
LIN {X 0,Y 478.289,Z 1152.36,A -85,B 0,C 180,E1 13788.91,E2 13788.91} C_VEL
